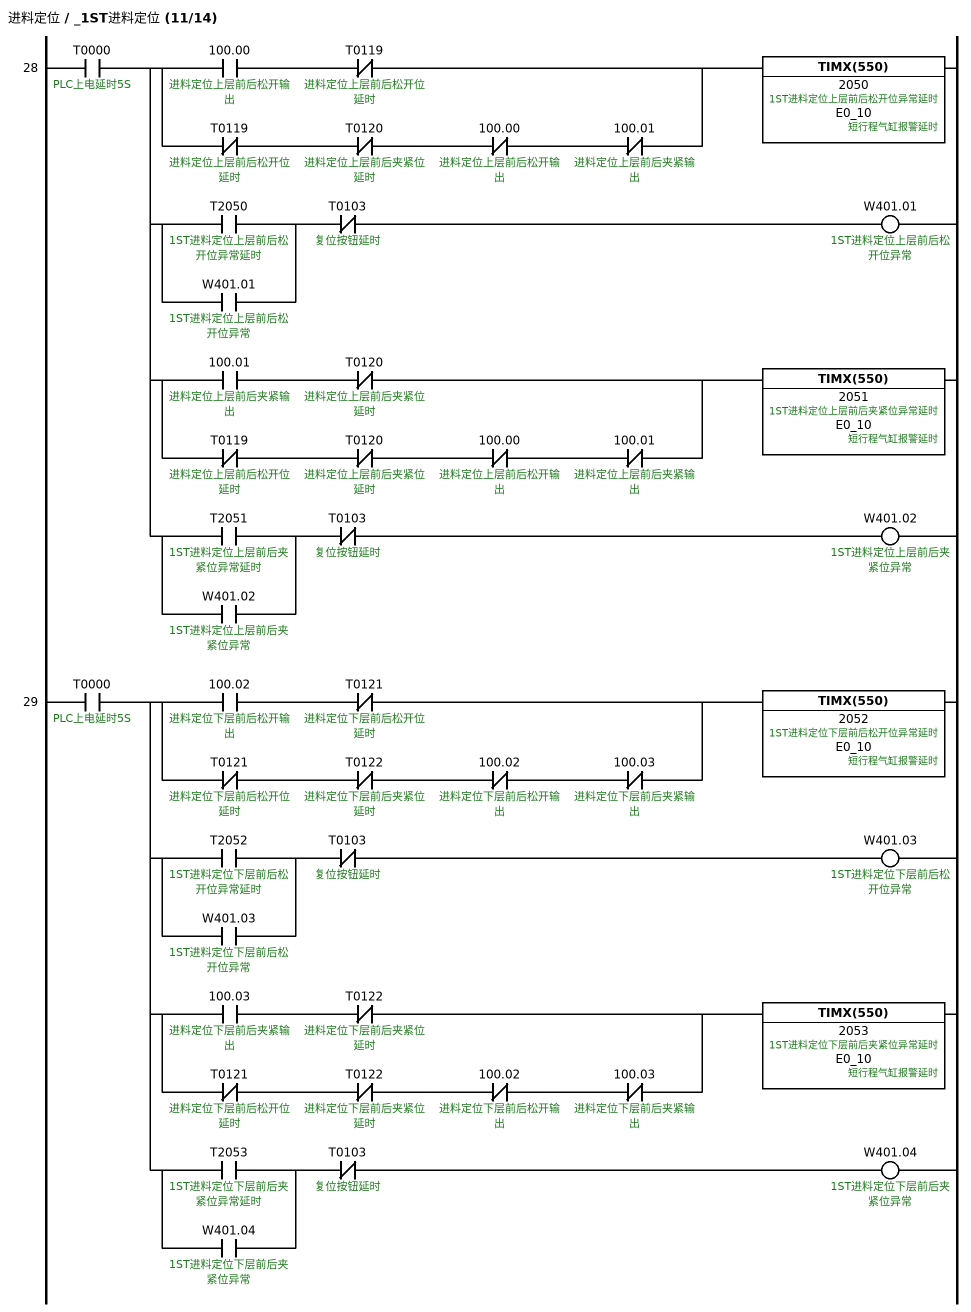
; [picture p72: 进料定位 / _1ST进料定位, rungs 28-29]
; rung 28
LD T0000  ; PLC上电延时5S
OUT TR0
LD 100.00  ; 进料定位上层前后松开输出
ANDNOT T0119  ; 进料定位上层前后松开位延时
LDNOT T0119  ; 进料定位上层前后松开位延时
ANDNOT T0120  ; 进料定位上层前后夹紧位延时
ANDNOT 100.00  ; 进料定位上层前后松开输出
ANDNOT 100.01  ; 进料定位上层前后夹紧输出
ORLD
ANDLD
TIMX(550) 2050 E0_10  ; 短行程气缸报警延时, 1ST进料定位上层前后松开位异常延时
LD TR0
LD T2050  ; 1ST进料定位上层前后松开位异常延时
OR W401.01  ; 1ST进料定位上层前后松开位异常
ANDLD
ANDNOT T0103  ; 复位按钮延时
OUT W401.01  ; 1ST进料定位上层前后松开位异常
LD TR0
LD 100.01  ; 进料定位上层前后夹紧输出
ANDNOT T0120  ; 进料定位上层前后夹紧位延时
LDNOT T0119  ; 进料定位上层前后松开位延时
ANDNOT T0120  ; 进料定位上层前后夹紧位延时
ANDNOT 100.00  ; 进料定位上层前后松开输出
ANDNOT 100.01  ; 进料定位上层前后夹紧输出
ORLD
ANDLD
TIMX(550) 2051 E0_10  ; 短行程气缸报警延时, 1ST进料定位上层前后夹紧位异常延时
LD TR0
LD T2051  ; 1ST进料定位上层前后夹紧位异常延时
OR W401.02  ; 1ST进料定位上层前后夹紧位异常
ANDLD
ANDNOT T0103  ; 复位按钮延时
OUT W401.02  ; 1ST进料定位上层前后夹紧位异常
; rung 29
LD T0000  ; PLC上电延时5S
OUT TR0
LD 100.02  ; 进料定位下层前后松开输出
ANDNOT T0121  ; 进料定位下层前后松开位延时
LDNOT T0121  ; 进料定位下层前后松开位延时
ANDNOT T0122  ; 进料定位下层前后夹紧位延时
ANDNOT 100.02  ; 进料定位下层前后松开输出
ANDNOT 100.03  ; 进料定位下层前后夹紧输出
ORLD
ANDLD
TIMX(550) 2052 E0_10  ; 短行程气缸报警延时, 1ST进料定位下层前后松开位异常延时
LD TR0
LD T2052  ; 1ST进料定位下层前后松开位异常延时
OR W401.03  ; 1ST进料定位下层前后松开位异常
ANDLD
ANDNOT T0103  ; 复位按钮延时
OUT W401.03  ; 1ST进料定位下层前后松开位异常
LD TR0
LD 100.03  ; 进料定位下层前后夹紧输出
ANDNOT T0122  ; 进料定位下层前后夹紧位延时
LDNOT T0121  ; 进料定位下层前后松开位延时
ANDNOT T0122  ; 进料定位下层前后夹紧位延时
ANDNOT 100.02  ; 进料定位下层前后松开输出
ANDNOT 100.03  ; 进料定位下层前后夹紧输出
ORLD
ANDLD
TIMX(550) 2053 E0_10  ; 短行程气缸报警延时, 1ST进料定位下层前后夹紧位异常延时
LD TR0
LD T2053  ; 1ST进料定位下层前后夹紧位异常延时
OR W401.04  ; 1ST进料定位下层前后夹紧位异常
ANDLD
ANDNOT T0103  ; 复位按钮延时
OUT W401.04  ; 1ST进料定位下层前后夹紧位异常

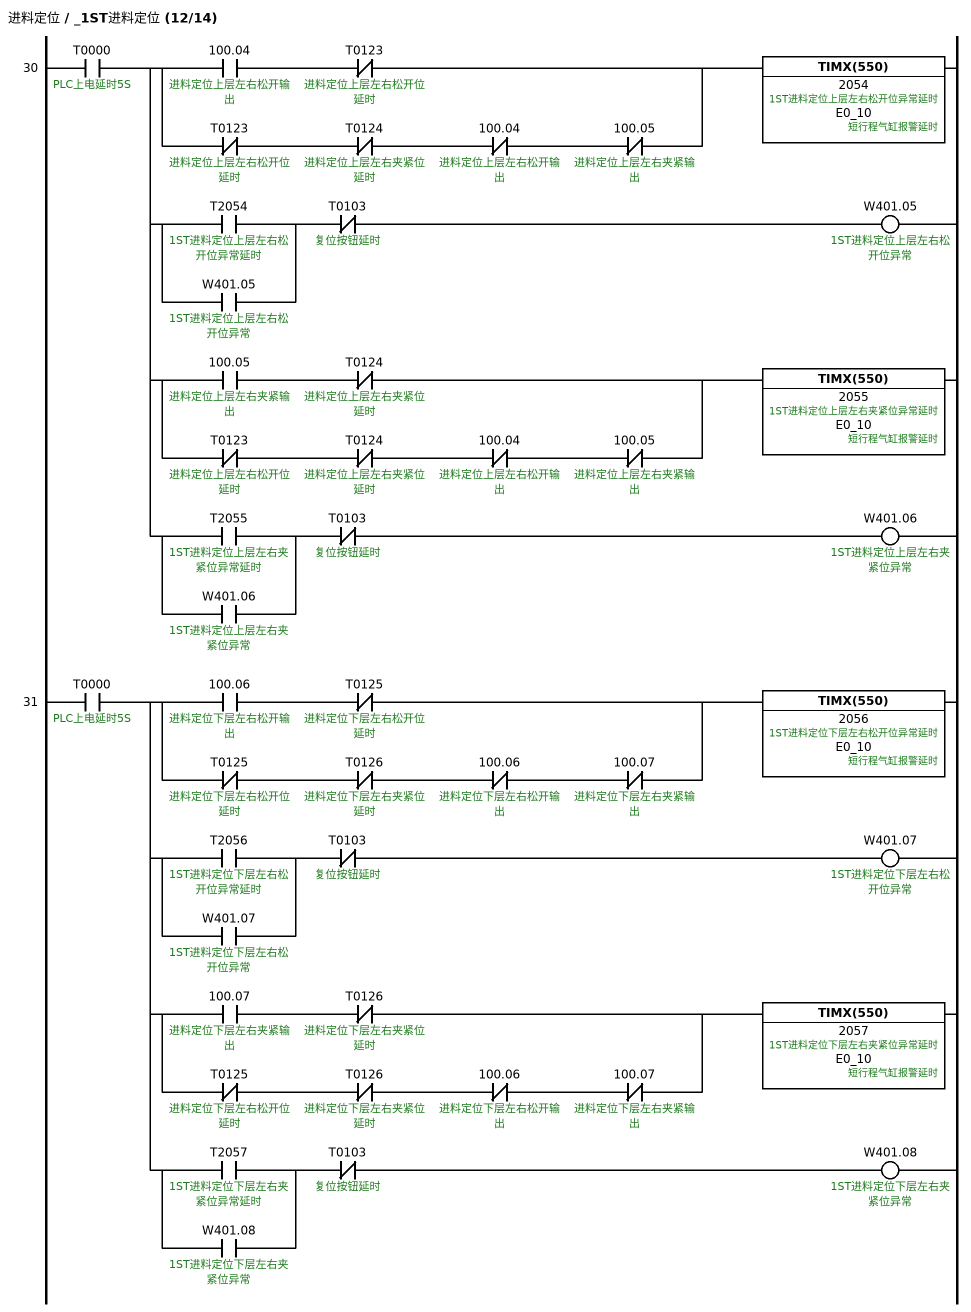
; rung 30
LD T0000  ; PLC上电延时5S
OUT TR0
LD 100.04  ; 进料定位上层左右松开输出
ANDNOT T0123  ; 进料定位上层左右松开位延时
LDNOT T0123  ; 进料定位上层左右松开位延时
ANDNOT T0124  ; 进料定位上层左右夹紧位延时
ANDNOT 100.04  ; 进料定位上层左右松开输出
ANDNOT 100.05  ; 进料定位上层左右夹紧输出
ORLD
ANDLD
TIMX(550) 2054 E0_10  ; 短行程气缸报警延时, 1ST进料定位上层左右松开位异常延时
LD TR0
LD T2054  ; 1ST进料定位上层左右松开位异常延时
OR W401.05  ; 1ST进料定位上层左右松开位异常
ANDLD
ANDNOT T0103  ; 复位按钮延时
OUT W401.05  ; 1ST进料定位上层左右松开位异常
LD TR0
LD 100.05  ; 进料定位上层左右夹紧输出
ANDNOT T0124  ; 进料定位上层左右夹紧位延时
LDNOT T0123  ; 进料定位上层左右松开位延时
ANDNOT T0124  ; 进料定位上层左右夹紧位延时
ANDNOT 100.04  ; 进料定位上层左右松开输出
ANDNOT 100.05  ; 进料定位上层左右夹紧输出
ORLD
ANDLD
TIMX(550) 2055 E0_10  ; 短行程气缸报警延时, 1ST进料定位上层左右夹紧位异常延时
LD TR0
LD T2055  ; 1ST进料定位上层左右夹紧位异常延时
OR W401.06  ; 1ST进料定位上层左右夹紧位异常
ANDLD
ANDNOT T0103  ; 复位按钮延时
OUT W401.06  ; 1ST进料定位上层左右夹紧位异常
; rung 31
LD T0000  ; PLC上电延时5S
OUT TR0
LD 100.06  ; 进料定位下层左右松开输出
ANDNOT T0125  ; 进料定位下层左右松开位延时
LDNOT T0125  ; 进料定位下层左右松开位延时
ANDNOT T0126  ; 进料定位下层左右夹紧位延时
ANDNOT 100.06  ; 进料定位下层左右松开输出
ANDNOT 100.07  ; 进料定位下层左右夹紧输出
ORLD
ANDLD
TIMX(550) 2056 E0_10  ; 短行程气缸报警延时, 1ST进料定位下层左右松开位异常延时
LD TR0
LD T2056  ; 1ST进料定位下层左右松开位异常延时
OR W401.07  ; 1ST进料定位下层左右松开位异常
ANDLD
ANDNOT T0103  ; 复位按钮延时
OUT W401.07  ; 1ST进料定位下层左右松开位异常
LD TR0
LD 100.07  ; 进料定位下层左右夹紧输出
ANDNOT T0126  ; 进料定位下层左右夹紧位延时
LDNOT T0125  ; 进料定位下层左右松开位延时
ANDNOT T0126  ; 进料定位下层左右夹紧位延时
ANDNOT 100.06  ; 进料定位下层左右松开输出
ANDNOT 100.07  ; 进料定位下层左右夹紧输出
ORLD
ANDLD
TIMX(550) 2057 E0_10  ; 短行程气缸报警延时, 1ST进料定位下层左右夹紧位异常延时
LD TR0
LD T2057  ; 1ST进料定位下层左右夹紧位异常延时
OR W401.08  ; 1ST进料定位下层左右夹紧位异常
ANDLD
ANDNOT T0103  ; 复位按钮延时
OUT W401.08  ; 1ST进料定位下层左右夹紧位异常

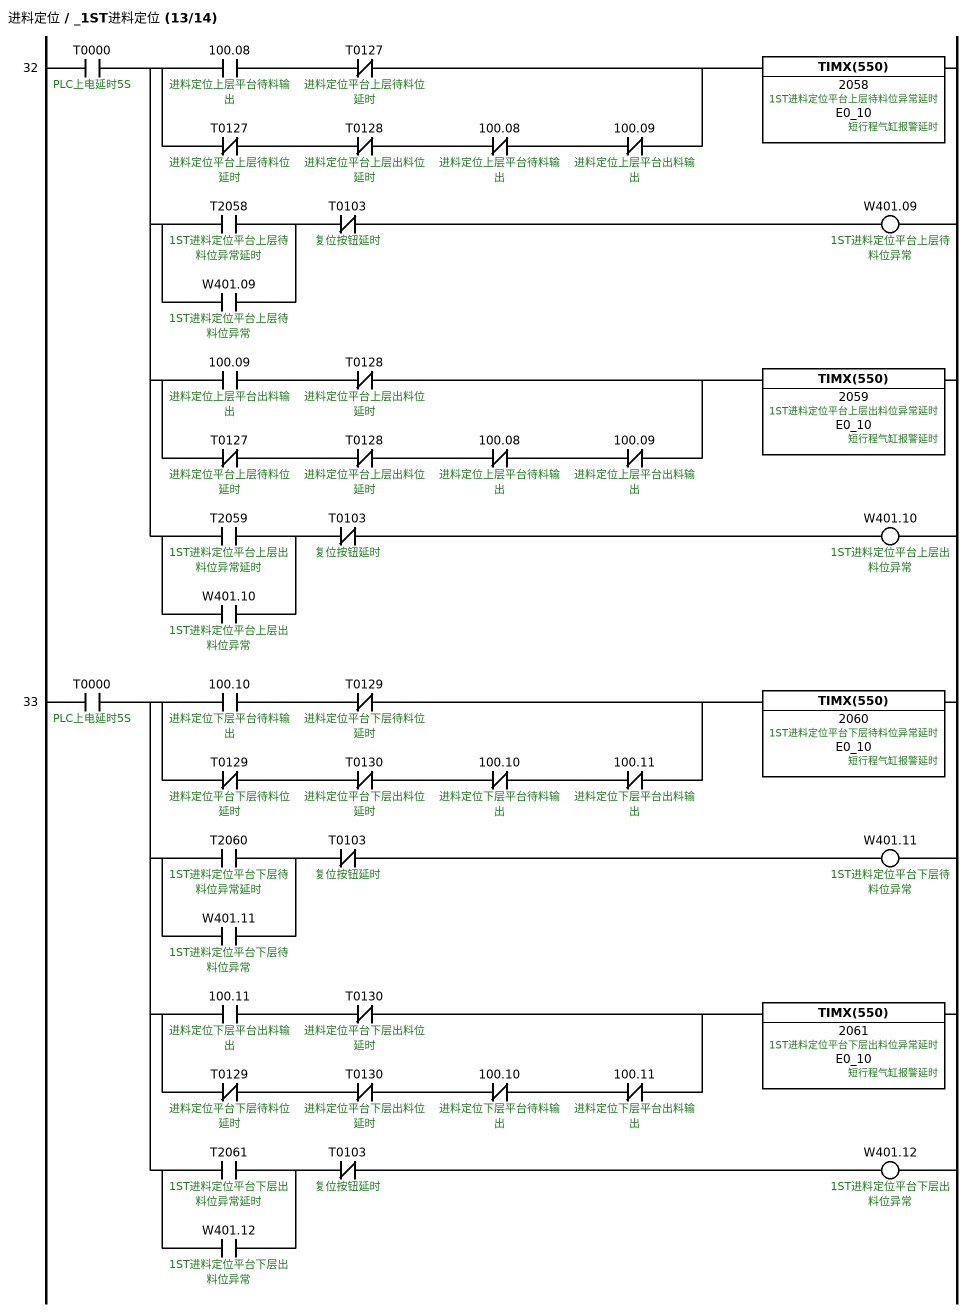
; rung 32
LD T0000  ; PLC上电延时5S
OUT TR0
LD 100.08  ; 进料定位上层平台待料输出
ANDNOT T0127  ; 进料定位平台上层待料位延时
LDNOT T0127  ; 进料定位平台上层待料位延时
ANDNOT T0128  ; 进料定位平台上层出料位延时
ANDNOT 100.08  ; 进料定位上层平台待料输出
ANDNOT 100.09  ; 进料定位上层平台出料输出
ORLD
ANDLD
TIMX(550) 2058 E0_10  ; 短行程气缸报警延时, 1ST进料定位平台上层待料位异常延时
LD TR0
LD T2058  ; 1ST进料定位平台上层待料位异常延时
OR W401.09  ; 1ST进料定位平台上层待料位异常
ANDLD
ANDNOT T0103  ; 复位按钮延时
OUT W401.09  ; 1ST进料定位平台上层待料位异常
LD TR0
LD 100.09  ; 进料定位上层平台出料输出
ANDNOT T0128  ; 进料定位平台上层出料位延时
LDNOT T0127  ; 进料定位平台上层待料位延时
ANDNOT T0128  ; 进料定位平台上层出料位延时
ANDNOT 100.08  ; 进料定位上层平台待料输出
ANDNOT 100.09  ; 进料定位上层平台出料输出
ORLD
ANDLD
TIMX(550) 2059 E0_10  ; 短行程气缸报警延时, 1ST进料定位平台上层出料位异常延时
LD TR0
LD T2059  ; 1ST进料定位平台上层出料位异常延时
OR W401.10  ; 1ST进料定位平台上层出料位异常
ANDLD
ANDNOT T0103  ; 复位按钮延时
OUT W401.10  ; 1ST进料定位平台上层出料位异常
; rung 33
LD T0000  ; PLC上电延时5S
OUT TR0
LD 100.10  ; 进料定位下层平台待料输出
ANDNOT T0129  ; 进料定位平台下层待料位延时
LDNOT T0129  ; 进料定位平台下层待料位延时
ANDNOT T0130  ; 进料定位平台下层出料位延时
ANDNOT 100.10  ; 进料定位下层平台待料输出
ANDNOT 100.11  ; 进料定位下层平台出料输出
ORLD
ANDLD
TIMX(550) 2060 E0_10  ; 短行程气缸报警延时, 1ST进料定位平台下层待料位异常延时
LD TR0
LD T2060  ; 1ST进料定位平台下层待料位异常延时
OR W401.11  ; 1ST进料定位平台下层待料位异常
ANDLD
ANDNOT T0103  ; 复位按钮延时
OUT W401.11  ; 1ST进料定位平台下层待料位异常
LD TR0
LD 100.11  ; 进料定位下层平台出料输出
ANDNOT T0130  ; 进料定位平台下层出料位延时
LDNOT T0129  ; 进料定位平台下层待料位延时
ANDNOT T0130  ; 进料定位平台下层出料位延时
ANDNOT 100.10  ; 进料定位下层平台待料输出
ANDNOT 100.11  ; 进料定位下层平台出料输出
ORLD
ANDLD
TIMX(550) 2061 E0_10  ; 短行程气缸报警延时, 1ST进料定位平台下层出料位异常延时
LD TR0
LD T2061  ; 1ST进料定位平台下层出料位异常延时
OR W401.12  ; 1ST进料定位平台下层出料位异常
ANDLD
ANDNOT T0103  ; 复位按钮延时
OUT W401.12  ; 1ST进料定位平台下层出料位异常

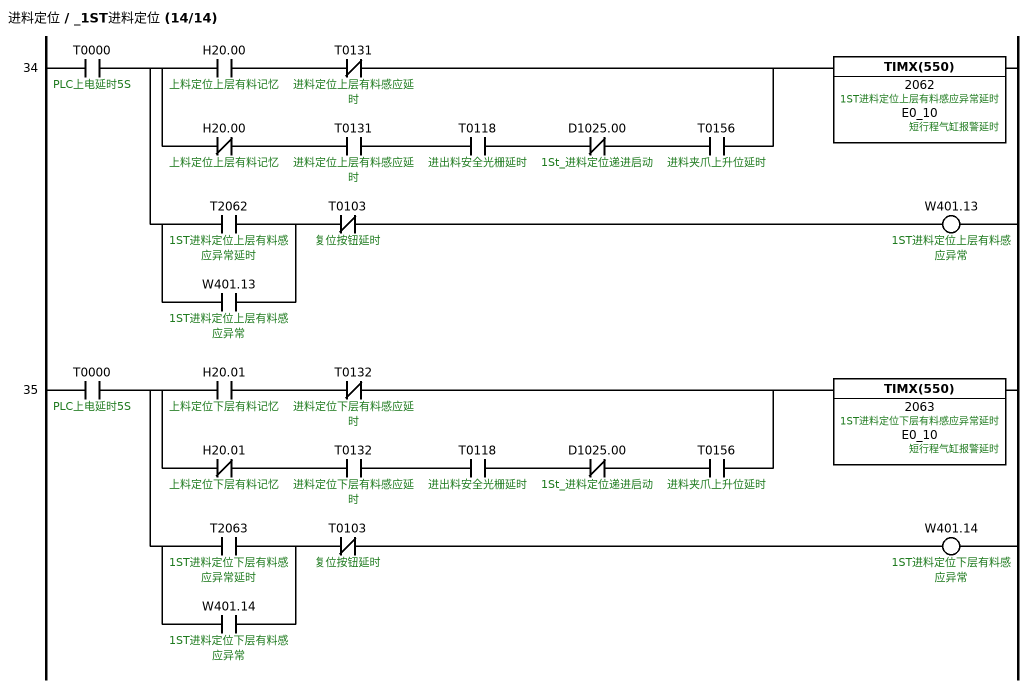
; rung 34
LD T0000  ; PLC上电延时5S
OUT TR0
LD H20.00  ; 上料定位上层有料记忆
ANDNOT T0131  ; 进料定位上层有料感应延时
LDNOT H20.00  ; 上料定位上层有料记忆
AND T0131  ; 进料定位上层有料感应延时
AND T0118  ; 进出料安全光栅延时
ANDNOT D1025.00  ; 1St_进料定位递进启动
AND T0156  ; 进料夹爪上升位延时
ORLD
ANDLD
TIMX(550) 2062 E0_10  ; 短行程气缸报警延时, 1ST进料定位上层有料感应异常延时
LD TR0
LD T2062  ; 1ST进料定位上层有料感应异常延时
OR W401.13  ; 1ST进料定位上层有料感应异常
ANDLD
ANDNOT T0103  ; 复位按钮延时
OUT W401.13  ; 1ST进料定位上层有料感应异常
; rung 35
LD T0000  ; PLC上电延时5S
OUT TR0
LD H20.01  ; 上料定位下层有料记忆
ANDNOT T0132  ; 进料定位下层有料感应延时
LDNOT H20.01  ; 上料定位下层有料记忆
AND T0132  ; 进料定位下层有料感应延时
AND T0118  ; 进出料安全光栅延时
ANDNOT D1025.00  ; 1St_进料定位递进启动
AND T0156  ; 进料夹爪上升位延时
ORLD
ANDLD
TIMX(550) 2063 E0_10  ; 短行程气缸报警延时, 1ST进料定位下层有料感应异常延时
LD TR0
LD T2063  ; 1ST进料定位下层有料感应异常延时
OR W401.14  ; 1ST进料定位下层有料感应异常
ANDLD
ANDNOT T0103  ; 复位按钮延时
OUT W401.14  ; 1ST进料定位下层有料感应异常

### Section 复位

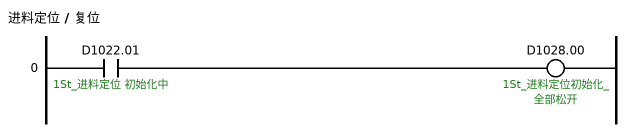
; rung 0
LD D1022.01  ; 1St_进料定位 初始化中
OUT D1028.00  ; 1St_进料定位初始化_全部松开

### Section 输出

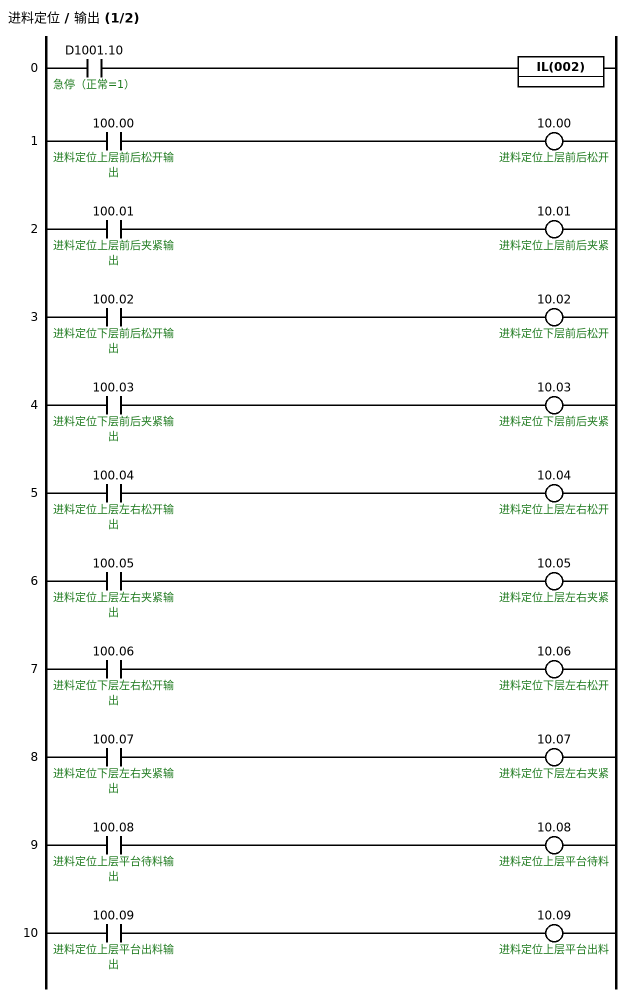
; rung 0
LD D1001.10  ; 急停（正常=1）
IL(002)
; rung 1
LD 100.00  ; 进料定位上层前后松开输出
OUT 10.00  ; 进料定位上层前后松开
; rung 2
LD 100.01  ; 进料定位上层前后夹紧输出
OUT 10.01  ; 进料定位上层前后夹紧
; rung 3
LD 100.02  ; 进料定位下层前后松开输出
OUT 10.02  ; 进料定位下层前后松开
; rung 4
LD 100.03  ; 进料定位下层前后夹紧输出
OUT 10.03  ; 进料定位下层前后夹紧
; rung 5
LD 100.04  ; 进料定位上层左右松开输出
OUT 10.04  ; 进料定位上层左右松开
; rung 6
LD 100.05  ; 进料定位上层左右夹紧输出
OUT 10.05  ; 进料定位上层左右夹紧
; rung 7
LD 100.06  ; 进料定位下层左右松开输出
OUT 10.06  ; 进料定位下层左右松开
; rung 8
LD 100.07  ; 进料定位下层左右夹紧输出
OUT 10.07  ; 进料定位下层左右夹紧
; rung 9
LD 100.08  ; 进料定位上层平台待料输出
OUT 10.08  ; 进料定位上层平台待料
; rung 10
LD 100.09  ; 进料定位上层平台出料输出
OUT 10.09  ; 进料定位上层平台出料

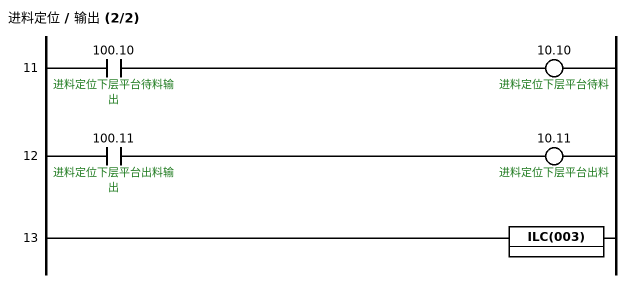
; rung 11
LD 100.10  ; 进料定位下层平台待料输出
OUT 10.10  ; 进料定位下层平台待料
; rung 12
LD 100.11  ; 进料定位下层平台出料输出
OUT 10.11  ; 进料定位下层平台出料
; rung 13
ILC(003)

### Section END
; rung 0
END(001)

## Program 出料定位 (cyclic task 2)

### Section Main

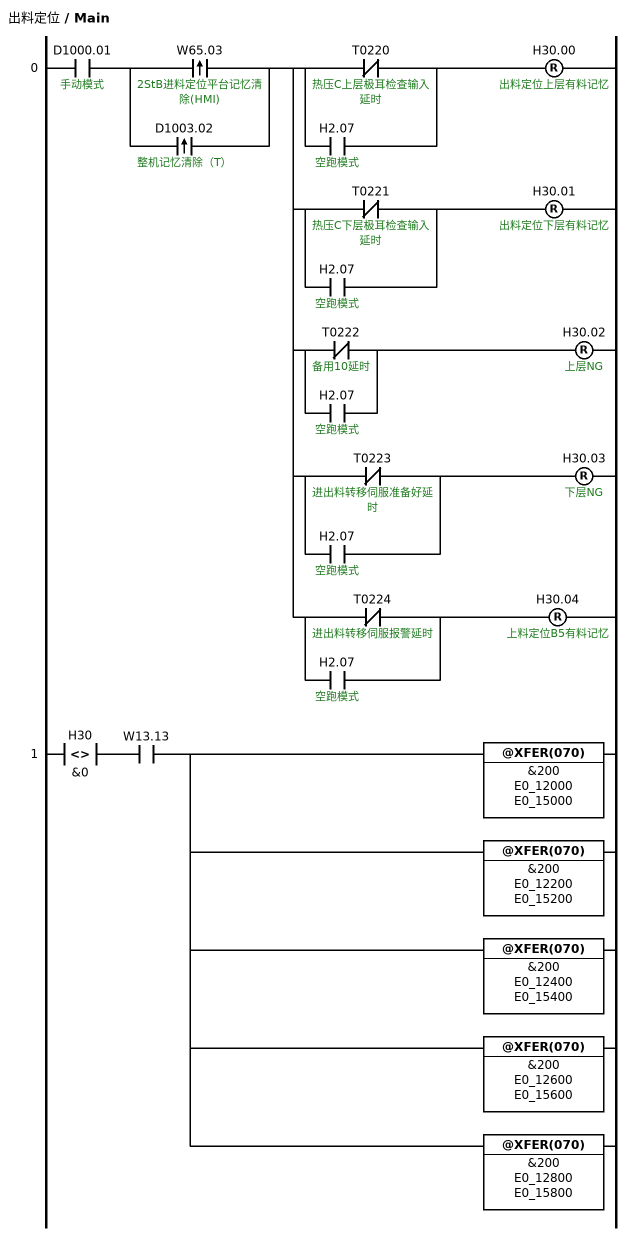
; rung 0
LD D1000.01  ; 手动模式
@LD W65.03  ; 2StB进料定位平台记忆清除(HMI)
@OR D1003.02  ; 整机记忆清除（T）
ANDLD
OUT TR0
LDNOT T0220  ; 热压C上层极耳检查输入延时
OR H2.07  ; 空跑模式
ANDLD
RSET H30.00  ; 出料定位上层有料记忆
LD TR0
LDNOT T0221  ; 热压C下层极耳检查输入延时
OR H2.07  ; 空跑模式
ANDLD
RSET H30.01  ; 出料定位下层有料记忆
LD TR0
LDNOT T0222  ; 备用10延时
OR H2.07  ; 空跑模式
ANDLD
RSET H30.02  ; 上层NG
LD TR0
LDNOT T0223  ; 进出料转移伺服准备好延时
OR H2.07  ; 空跑模式
ANDLD
RSET H30.03  ; 下层NG
LD TR0
LDNOT T0224  ; 进出料转移伺服报警延时
OR H2.07  ; 空跑模式
ANDLD
RSET H30.04  ; 上料定位B5有料记忆
; rung 1
LD<>(305) H30 &0
AND W13.13
@XFER(070) &200 E0_12000 E0_15000
@XFER(070) &200 E0_12200 E0_15200
@XFER(070) &200 E0_12400 E0_15400
@XFER(070) &200 E0_12600 E0_15600
@XFER(070) &200 E0_12800 E0_15800

### Section _2ST出料定位

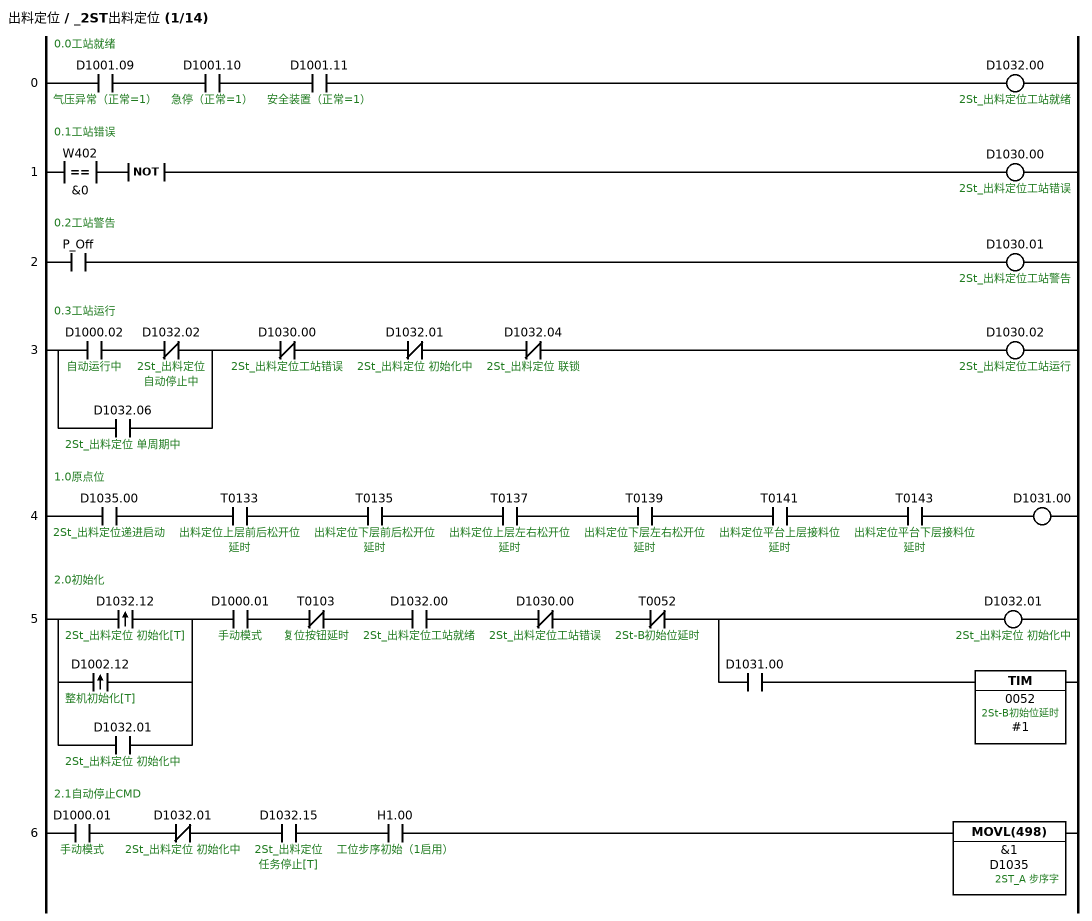
; rung 0: 0.0工站就绪
LD D1001.09  ; 气压异常（正常=1）
AND D1001.10  ; 急停（正常=1）
AND D1001.11  ; 安全装置（正常=1）
OUT D1032.00  ; 2St_出料定位工站就绪
; rung 1: 0.1工站错误
LD=(300) W402 &0
NOT(520)
OUT D1030.00  ; 2St_出料定位工站错误
; rung 2: 0.2工站警告
LD P_Off
OUT D1030.01  ; 2St_出料定位工站警告
; rung 3: 0.3工站运行
LD D1000.02  ; 自动运行中
ANDNOT D1032.02  ; 2St_出料定位 自动停止中
OR D1032.06  ; 2St_出料定位 单周期中
ANDNOT D1030.00  ; 2St_出料定位工站错误
ANDNOT D1032.01  ; 2St_出料定位 初始化中
ANDNOT D1032.04  ; 2St_出料定位 联锁
OUT D1030.02  ; 2St_出料定位工站运行
; rung 4: 1.0原点位
LD D1035.00  ; 2St_出料定位递进启动
AND T0133  ; 出料定位上层前后松开位延时
AND T0135  ; 出料定位下层前后松开位延时
AND T0137  ; 出料定位上层左右松开位延时
AND T0139  ; 出料定位下层左右松开位延时
AND T0141  ; 出料定位平台上层接料位延时
AND T0143  ; 出料定位平台下层接料位延时
OUT D1031.00
; rung 5: 2.0初始化
@LD D1032.12  ; 2St_出料定位 初始化[T]
@OR D1002.12  ; 整机初始化[T]
OR D1032.01  ; 2St_出料定位 初始化中
AND D1000.01  ; 手动模式
ANDNOT T0103  ; 复位按钮延时
AND D1032.00  ; 2St_出料定位工站就绪
ANDNOT D1030.00  ; 2St_出料定位工站错误
ANDNOT T0052  ; 2St-B初始位延时
OUT D1032.01  ; 2St_出料定位 初始化中
AND D1031.00
TIM 0052 #1  ; 2St-B初始位延时
; rung 6: 2.1自动停止CMD
LD D1000.01  ; 手动模式
ANDNOT D1032.01  ; 2St_出料定位 初始化中
AND D1032.15  ; 2St_出料定位 任务停止[T]
AND H1.00  ; 工位步序初始（1启用）
MOVL(498) &1 D1035  ; 2ST_A 步序字

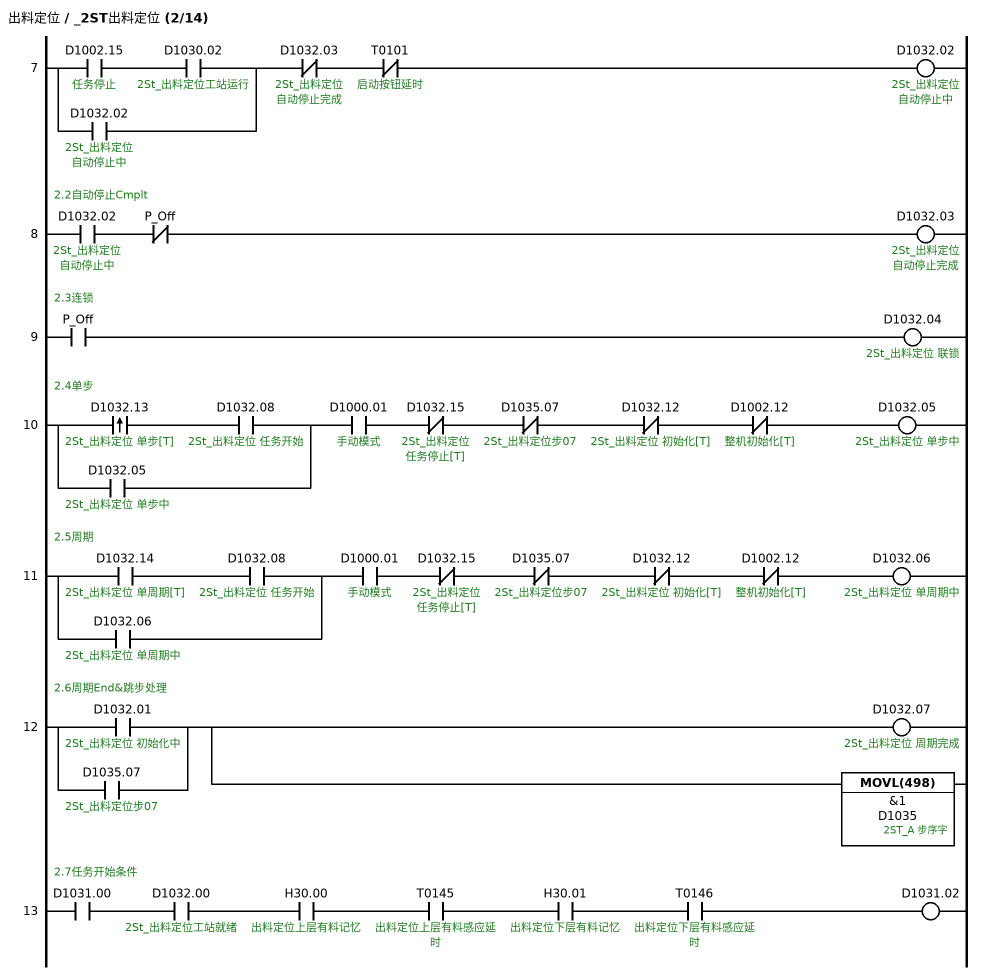
; rung 7
LD D1002.15  ; 任务停止
AND D1030.02  ; 2St_出料定位工站运行
OR D1032.02  ; 2St_出料定位 自动停止中
ANDNOT D1032.03  ; 2St_出料定位 自动停止完成
ANDNOT T0101  ; 启动按钮延时
OUT D1032.02  ; 2St_出料定位 自动停止中
; rung 8: 2.2自动停止Cmplt
LD D1032.02  ; 2St_出料定位 自动停止中
ANDNOT P_Off
OUT D1032.03  ; 2St_出料定位 自动停止完成
; rung 9: 2.3连锁
LD P_Off
OUT D1032.04  ; 2St_出料定位 联锁
; rung 10: 2.4单步
@LD D1032.13  ; 2St_出料定位 单步[T]
AND D1032.08  ; 2St_出料定位 任务开始
OR D1032.05  ; 2St_出料定位 单步中
AND D1000.01  ; 手动模式
ANDNOT D1032.15  ; 2St_出料定位 任务停止[T]
ANDNOT D1035.07  ; 2St_出料定位步07
ANDNOT D1032.12  ; 2St_出料定位 初始化[T]
ANDNOT D1002.12  ; 整机初始化[T]
OUT D1032.05  ; 2St_出料定位 单步中
; rung 11: 2.5周期
LD D1032.14  ; 2St_出料定位 单周期[T]
AND D1032.08  ; 2St_出料定位 任务开始
OR D1032.06  ; 2St_出料定位 单周期中
AND D1000.01  ; 手动模式
ANDNOT D1032.15  ; 2St_出料定位 任务停止[T]
ANDNOT D1035.07  ; 2St_出料定位步07
ANDNOT D1032.12  ; 2St_出料定位 初始化[T]
ANDNOT D1002.12  ; 整机初始化[T]
OUT D1032.06  ; 2St_出料定位 单周期中
; rung 12: 2.6周期End&跳步处理
LD D1032.01  ; 2St_出料定位 初始化中
OR D1035.07  ; 2St_出料定位步07
OUT D1032.07  ; 2St_出料定位 周期完成
MOVL(498) &1 D1035  ; 2ST_A 步序字
; rung 13: 2.7任务开始条件
LD D1031.00
AND D1032.00  ; 2St_出料定位工站就绪
AND H30.00  ; 出料定位上层有料记忆
AND T0145  ; 出料定位上层有料感应延时
AND H30.01  ; 出料定位下层有料记忆
AND T0146  ; 出料定位下层有料感应延时
OUT D1031.02

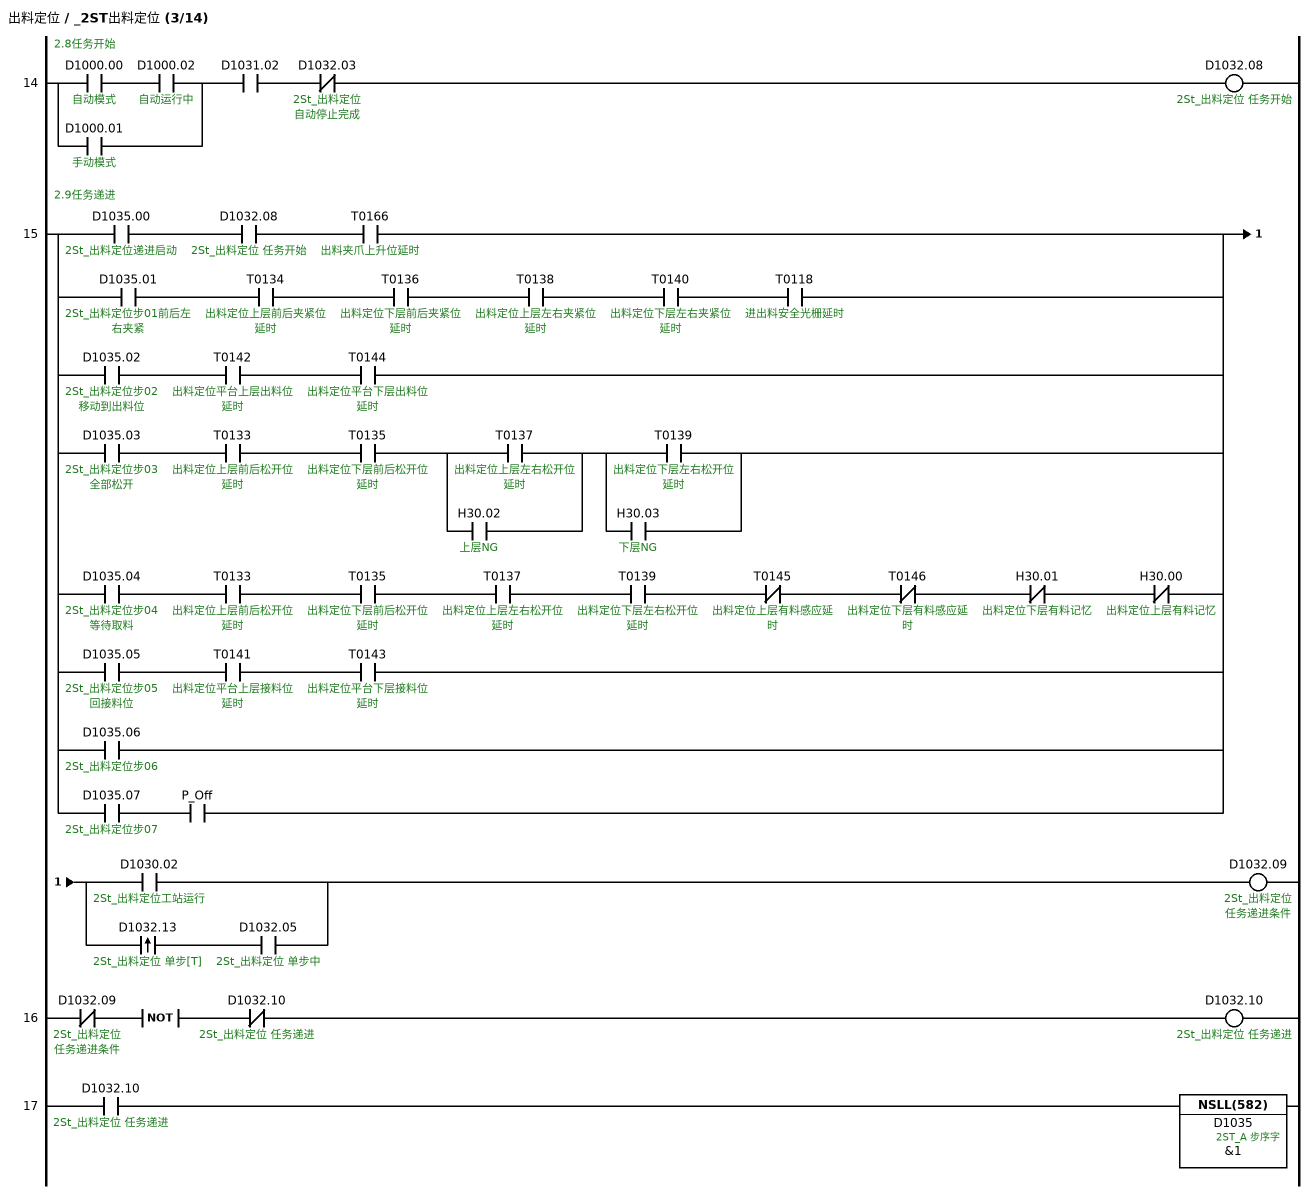
; rung 14: 2.8任务开始
LD D1000.00  ; 自动模式
AND D1000.02  ; 自动运行中
OR D1000.01  ; 手动模式
AND D1031.02
ANDNOT D1032.03  ; 2St_出料定位 自动停止完成
OUT D1032.08  ; 2St_出料定位 任务开始
; rung 15: 2.9任务递进
LD D1035.00  ; 2St_出料定位递进启动
AND D1032.08  ; 2St_出料定位 任务开始
AND T0166  ; 出料夹爪上升位延时
LD D1035.01  ; 2St_出料定位步01前后左右夹紧
AND T0134  ; 出料定位上层前后夹紧位延时
AND T0136  ; 出料定位下层前后夹紧位延时
AND T0138  ; 出料定位上层左右夹紧位延时
AND T0140  ; 出料定位下层左右夹紧位延时
AND T0118  ; 进出料安全光栅延时
ORLD
LD D1035.02  ; 2St_出料定位步02 移动到出料位
AND T0142  ; 出料定位平台上层出料位延时
AND T0144  ; 出料定位平台下层出料位延时
ORLD
LD D1035.03  ; 2St_出料定位步03 全部松开
AND T0133  ; 出料定位上层前后松开位延时
AND T0135  ; 出料定位下层前后松开位延时
LD T0137  ; 出料定位上层左右松开位延时
OR H30.02  ; 上层NG
ANDLD
LD T0139  ; 出料定位下层左右松开位延时
OR H30.03  ; 下层NG
ANDLD
ORLD
LD D1035.04  ; 2St_出料定位步04 等待取料
AND T0133  ; 出料定位上层前后松开位延时
AND T0135  ; 出料定位下层前后松开位延时
AND T0137  ; 出料定位上层左右松开位延时
AND T0139  ; 出料定位下层左右松开位延时
ANDNOT T0145  ; 出料定位上层有料感应延时
ANDNOT T0146  ; 出料定位下层有料感应延时
ANDNOT H30.01  ; 出料定位下层有料记忆
ANDNOT H30.00  ; 出料定位上层有料记忆
ORLD
LD D1035.05  ; 2St_出料定位步05 回接料位
AND T0141  ; 出料定位平台上层接料位延时
AND T0143  ; 出料定位平台下层接料位延时
ORLD
OR D1035.06  ; 2St_出料定位步06
LD D1035.07  ; 2St_出料定位步07
AND P_Off
ORLD
LD D1030.02  ; 2St_出料定位工站运行
@LD D1032.13  ; 2St_出料定位 单步[T]
AND D1032.05  ; 2St_出料定位 单步中
ORLD
ANDLD
OUT D1032.09  ; 2St_出料定位 任务递进条件
; rung 16
LDNOT D1032.09  ; 2St_出料定位 任务递进条件
NOT(520)
ANDNOT D1032.10  ; 2St_出料定位 任务递进
OUT D1032.10  ; 2St_出料定位 任务递进
; rung 17
LD D1032.10  ; 2St_出料定位 任务递进
NSLL(582) D1035 &1  ; 2ST_A 步序字

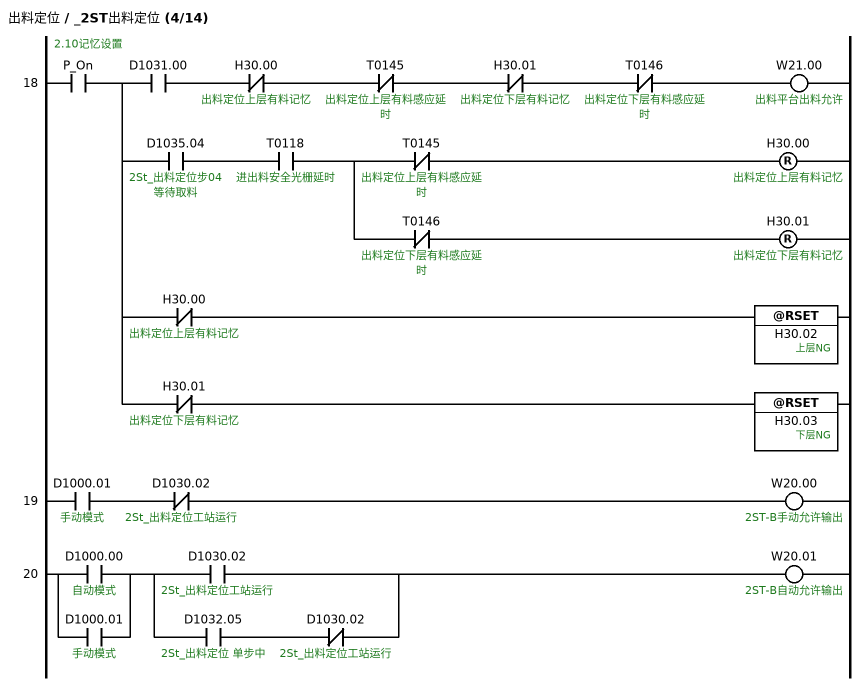
; rung 18: 2.10记忆设置
LD P_On
OUT TR0
AND D1031.00
ANDNOT H30.00  ; 出料定位上层有料记忆
ANDNOT T0145  ; 出料定位上层有料感应延时
ANDNOT H30.01  ; 出料定位下层有料记忆
ANDNOT T0146  ; 出料定位下层有料感应延时
OUT W21.00  ; 出料平台出料允许
LD TR0
AND D1035.04  ; 2St_出料定位步04 等待取料
AND T0118  ; 进出料安全光栅延时
OUT TR1
ANDNOT T0145  ; 出料定位上层有料感应延时
RSET H30.00  ; 出料定位上层有料记忆
LD TR1
ANDNOT T0146  ; 出料定位下层有料感应延时
RSET H30.01  ; 出料定位下层有料记忆
LD TR0
ANDNOT H30.00  ; 出料定位上层有料记忆
@RSET H30.02  ; 上层NG
LD TR0
ANDNOT H30.01  ; 出料定位下层有料记忆
@RSET H30.03  ; 下层NG
; rung 19
LD D1000.01  ; 手动模式
ANDNOT D1030.02  ; 2St_出料定位工站运行
OUT W20.00  ; 2ST-B手动允许输出
; rung 20
LD D1000.00  ; 自动模式
OR D1000.01  ; 手动模式
LD D1030.02  ; 2St_出料定位工站运行
LD D1032.05  ; 2St_出料定位 单步中
ANDNOT D1030.02  ; 2St_出料定位工站运行
ORLD
ANDLD
OUT W20.01  ; 2ST-B自动允许输出

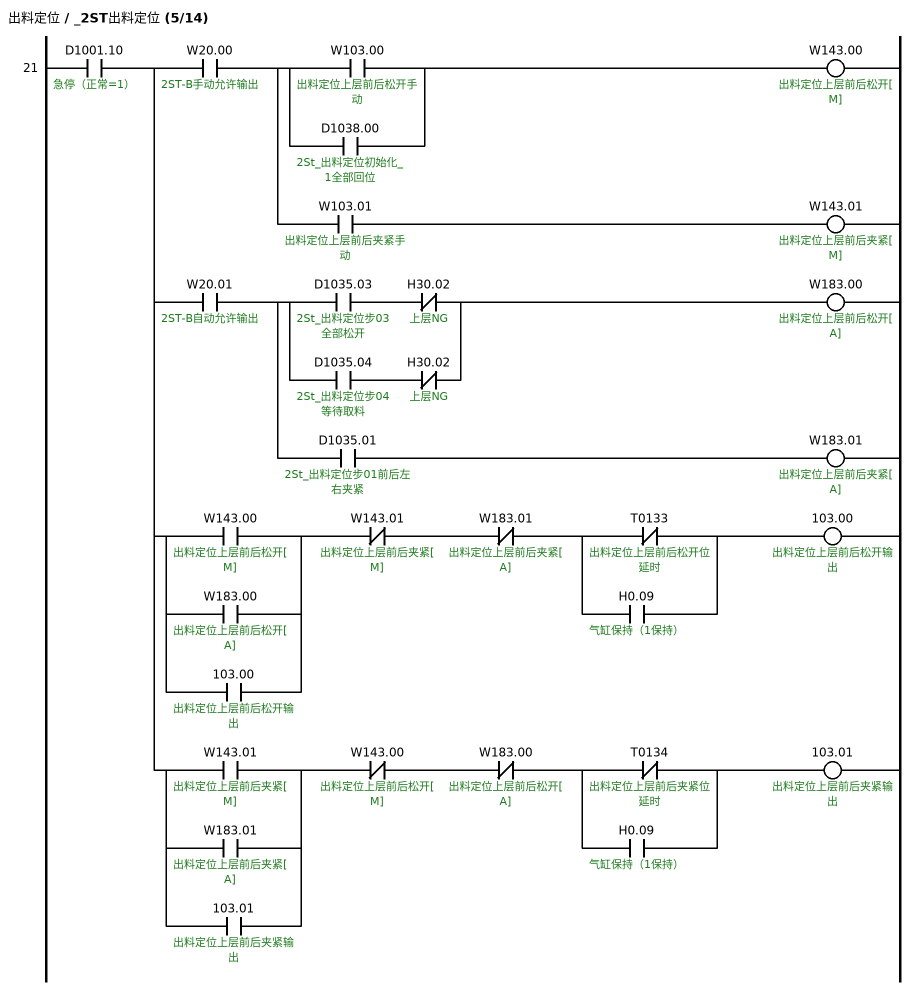
; rung 21
LD D1001.10  ; 急停（正常=1）
OUT TR0
AND W20.00  ; 2ST-B手动允许输出
OUT TR1
LD W103.00  ; 出料定位上层前后松开手动
OR D1038.00  ; 2St_出料定位初始化_1全部回位
ANDLD
OUT W143.00  ; 出料定位上层前后松开[M]
LD TR1
AND W103.01  ; 出料定位上层前后夹紧手动
OUT W143.01  ; 出料定位上层前后夹紧[M]
LD TR0
AND W20.01  ; 2ST-B自动允许输出
OUT TR1
LD D1035.03  ; 2St_出料定位步03 全部松开
ANDNOT H30.02  ; 上层NG
LD D1035.04  ; 2St_出料定位步04 等待取料
ANDNOT H30.02  ; 上层NG
ORLD
ANDLD
OUT W183.00  ; 出料定位上层前后松开[A]
LD TR1
AND D1035.01  ; 2St_出料定位步01前后左右夹紧
OUT W183.01  ; 出料定位上层前后夹紧[A]
LD TR0
LD W143.00  ; 出料定位上层前后松开[M]
OR W183.00  ; 出料定位上层前后松开[A]
OR 103.00  ; 出料定位上层前后松开输出
ANDLD
ANDNOT W143.01  ; 出料定位上层前后夹紧[M]
ANDNOT W183.01  ; 出料定位上层前后夹紧[A]
LDNOT T0133  ; 出料定位上层前后松开位延时
OR H0.09  ; 气缸保持（1保持）
ANDLD
OUT 103.00  ; 出料定位上层前后松开输出
LD TR0
LD W143.01  ; 出料定位上层前后夹紧[M]
OR W183.01  ; 出料定位上层前后夹紧[A]
OR 103.01  ; 出料定位上层前后夹紧输出
ANDLD
ANDNOT W143.00  ; 出料定位上层前后松开[M]
ANDNOT W183.00  ; 出料定位上层前后松开[A]
LDNOT T0134  ; 出料定位上层前后夹紧位延时
OR H0.09  ; 气缸保持（1保持）
ANDLD
OUT 103.01  ; 出料定位上层前后夹紧输出

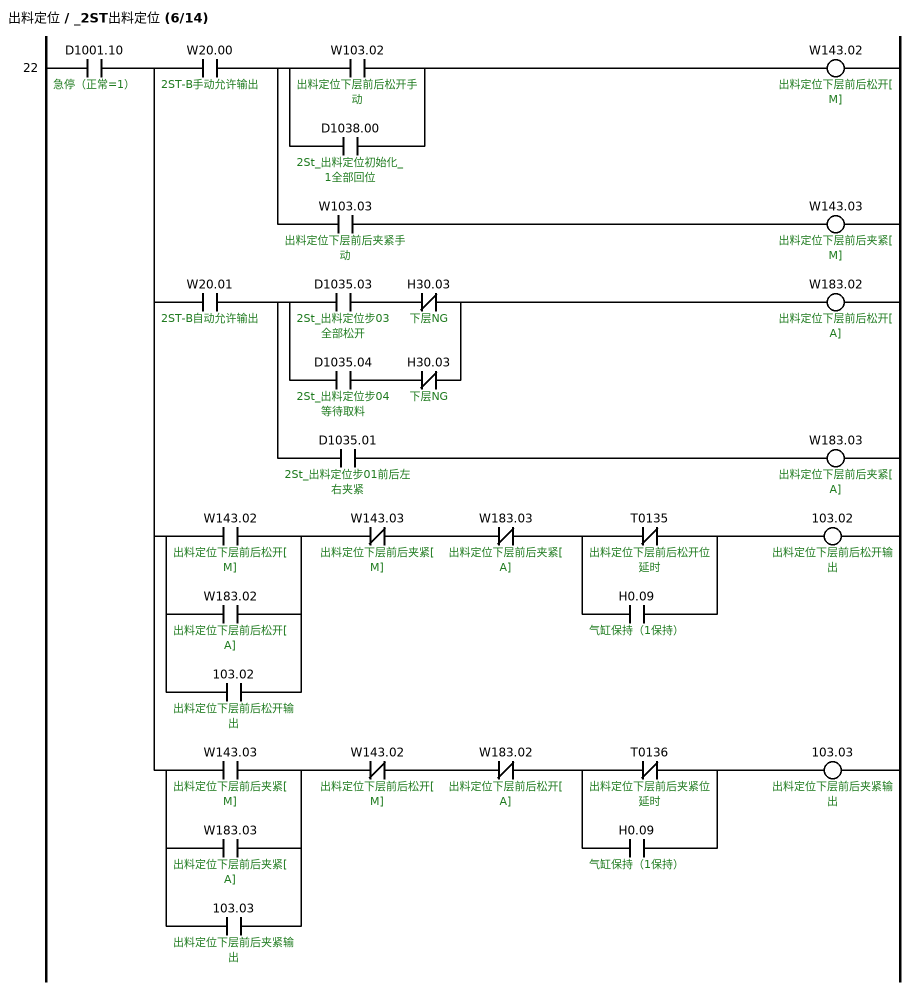
; rung 22
LD D1001.10  ; 急停（正常=1）
OUT TR0
AND W20.00  ; 2ST-B手动允许输出
OUT TR1
LD W103.02  ; 出料定位下层前后松开手动
OR D1038.00  ; 2St_出料定位初始化_1全部回位
ANDLD
OUT W143.02  ; 出料定位下层前后松开[M]
LD TR1
AND W103.03  ; 出料定位下层前后夹紧手动
OUT W143.03  ; 出料定位下层前后夹紧[M]
LD TR0
AND W20.01  ; 2ST-B自动允许输出
OUT TR1
LD D1035.03  ; 2St_出料定位步03 全部松开
ANDNOT H30.03  ; 下层NG
LD D1035.04  ; 2St_出料定位步04 等待取料
ANDNOT H30.03  ; 下层NG
ORLD
ANDLD
OUT W183.02  ; 出料定位下层前后松开[A]
LD TR1
AND D1035.01  ; 2St_出料定位步01前后左右夹紧
OUT W183.03  ; 出料定位下层前后夹紧[A]
LD TR0
LD W143.02  ; 出料定位下层前后松开[M]
OR W183.02  ; 出料定位下层前后松开[A]
OR 103.02  ; 出料定位下层前后松开输出
ANDLD
ANDNOT W143.03  ; 出料定位下层前后夹紧[M]
ANDNOT W183.03  ; 出料定位下层前后夹紧[A]
LDNOT T0135  ; 出料定位下层前后松开位延时
OR H0.09  ; 气缸保持（1保持）
ANDLD
OUT 103.02  ; 出料定位下层前后松开输出
LD TR0
LD W143.03  ; 出料定位下层前后夹紧[M]
OR W183.03  ; 出料定位下层前后夹紧[A]
OR 103.03  ; 出料定位下层前后夹紧输出
ANDLD
ANDNOT W143.02  ; 出料定位下层前后松开[M]
ANDNOT W183.02  ; 出料定位下层前后松开[A]
LDNOT T0136  ; 出料定位下层前后夹紧位延时
OR H0.09  ; 气缸保持（1保持）
ANDLD
OUT 103.03  ; 出料定位下层前后夹紧输出

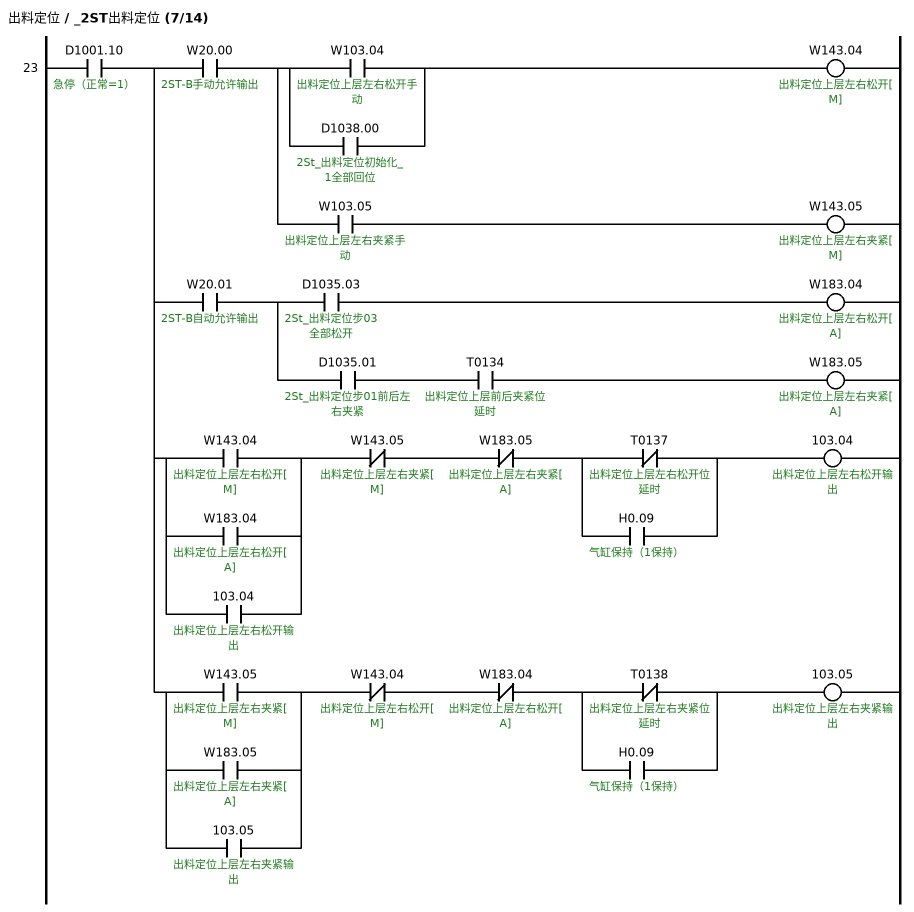
; rung 23
LD D1001.10  ; 急停（正常=1）
OUT TR0
AND W20.00  ; 2ST-B手动允许输出
OUT TR1
LD W103.04  ; 出料定位上层左右松开手动
OR D1038.00  ; 2St_出料定位初始化_1全部回位
ANDLD
OUT W143.04  ; 出料定位上层左右松开[M]
LD TR1
AND W103.05  ; 出料定位上层左右夹紧手动
OUT W143.05  ; 出料定位上层左右夹紧[M]
LD TR0
AND W20.01  ; 2ST-B自动允许输出
OUT TR1
AND D1035.03  ; 2St_出料定位步03 全部松开
OUT W183.04  ; 出料定位上层左右松开[A]
LD TR1
AND D1035.01  ; 2St_出料定位步01前后左右夹紧
AND T0134  ; 出料定位上层前后夹紧位延时
OUT W183.05  ; 出料定位上层左右夹紧[A]
LD TR0
LD W143.04  ; 出料定位上层左右松开[M]
OR W183.04  ; 出料定位上层左右松开[A]
OR 103.04  ; 出料定位上层左右松开输出
ANDLD
ANDNOT W143.05  ; 出料定位上层左右夹紧[M]
ANDNOT W183.05  ; 出料定位上层左右夹紧[A]
LDNOT T0137  ; 出料定位上层左右松开位延时
OR H0.09  ; 气缸保持（1保持）
ANDLD
OUT 103.04  ; 出料定位上层左右松开输出
LD TR0
LD W143.05  ; 出料定位上层左右夹紧[M]
OR W183.05  ; 出料定位上层左右夹紧[A]
OR 103.05  ; 出料定位上层左右夹紧输出
ANDLD
ANDNOT W143.04  ; 出料定位上层左右松开[M]
ANDNOT W183.04  ; 出料定位上层左右松开[A]
LDNOT T0138  ; 出料定位上层左右夹紧位延时
OR H0.09  ; 气缸保持（1保持）
ANDLD
OUT 103.05  ; 出料定位上层左右夹紧输出

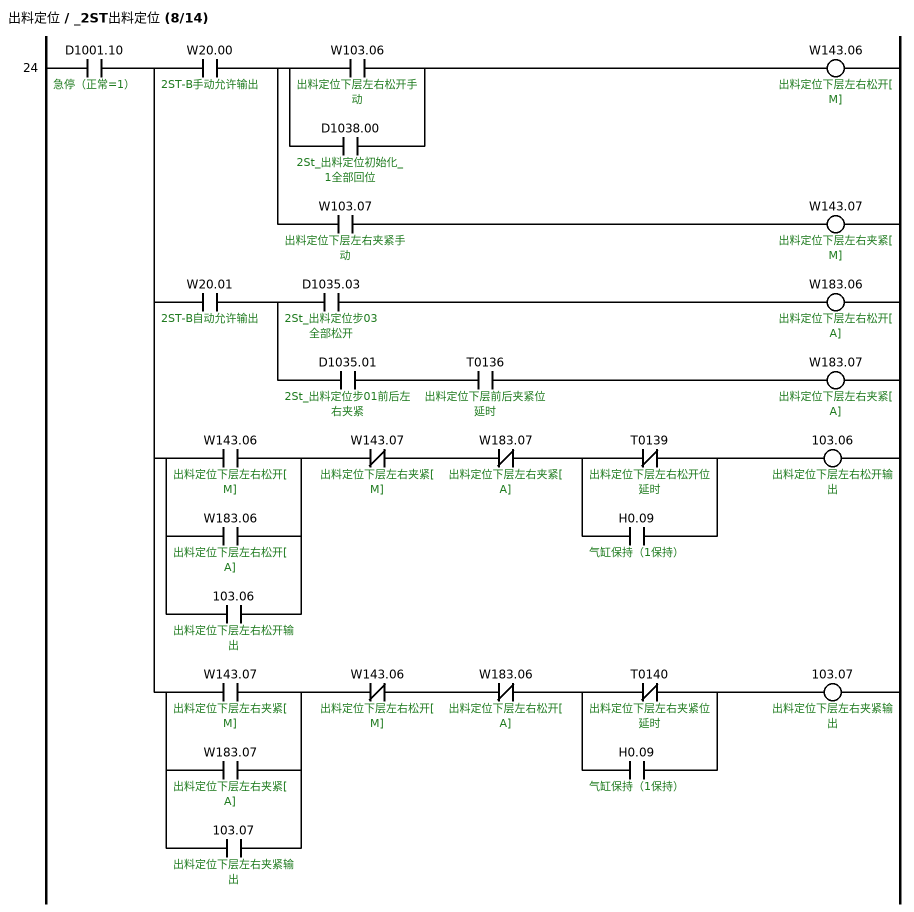
; rung 24
LD D1001.10  ; 急停（正常=1）
OUT TR0
AND W20.00  ; 2ST-B手动允许输出
OUT TR1
LD W103.06  ; 出料定位下层左右松开手动
OR D1038.00  ; 2St_出料定位初始化_1全部回位
ANDLD
OUT W143.06  ; 出料定位下层左右松开[M]
LD TR1
AND W103.07  ; 出料定位下层左右夹紧手动
OUT W143.07  ; 出料定位下层左右夹紧[M]
LD TR0
AND W20.01  ; 2ST-B自动允许输出
OUT TR1
AND D1035.03  ; 2St_出料定位步03 全部松开
OUT W183.06  ; 出料定位下层左右松开[A]
LD TR1
AND D1035.01  ; 2St_出料定位步01前后左右夹紧
AND T0136  ; 出料定位下层前后夹紧位延时
OUT W183.07  ; 出料定位下层左右夹紧[A]
LD TR0
LD W143.06  ; 出料定位下层左右松开[M]
OR W183.06  ; 出料定位下层左右松开[A]
OR 103.06  ; 出料定位下层左右松开输出
ANDLD
ANDNOT W143.07  ; 出料定位下层左右夹紧[M]
ANDNOT W183.07  ; 出料定位下层左右夹紧[A]
LDNOT T0139  ; 出料定位下层左右松开位延时
OR H0.09  ; 气缸保持（1保持）
ANDLD
OUT 103.06  ; 出料定位下层左右松开输出
LD TR0
LD W143.07  ; 出料定位下层左右夹紧[M]
OR W183.07  ; 出料定位下层左右夹紧[A]
OR 103.07  ; 出料定位下层左右夹紧输出
ANDLD
ANDNOT W143.06  ; 出料定位下层左右松开[M]
ANDNOT W183.06  ; 出料定位下层左右松开[A]
LDNOT T0140  ; 出料定位下层左右夹紧位延时
OR H0.09  ; 气缸保持（1保持）
ANDLD
OUT 103.07  ; 出料定位下层左右夹紧输出

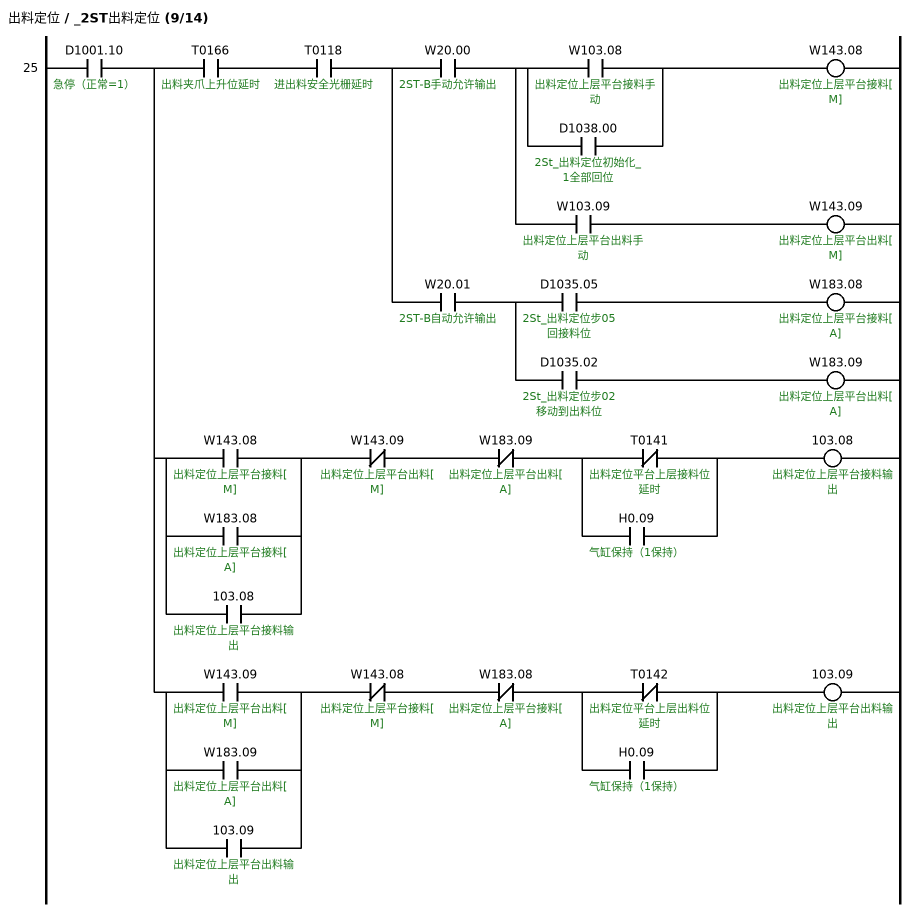
; rung 25
LD D1001.10  ; 急停（正常=1）
OUT TR0
AND T0166  ; 出料夹爪上升位延时
AND T0118  ; 进出料安全光栅延时
OUT TR1
AND W20.00  ; 2ST-B手动允许输出
OUT TR2
LD W103.08  ; 出料定位上层平台接料手动
OR D1038.00  ; 2St_出料定位初始化_1全部回位
ANDLD
OUT W143.08  ; 出料定位上层平台接料[M]
LD TR2
AND W103.09  ; 出料定位上层平台出料手动
OUT W143.09  ; 出料定位上层平台出料[M]
LD TR1
AND W20.01  ; 2ST-B自动允许输出
OUT TR1
AND D1035.05  ; 2St_出料定位步05 回接料位
OUT W183.08  ; 出料定位上层平台接料[A]
LD TR1
AND D1035.02  ; 2St_出料定位步02 移动到出料位
OUT W183.09  ; 出料定位上层平台出料[A]
LD TR0
LD W143.08  ; 出料定位上层平台接料[M]
OR W183.08  ; 出料定位上层平台接料[A]
OR 103.08  ; 出料定位上层平台接料输出
ANDLD
ANDNOT W143.09  ; 出料定位上层平台出料[M]
ANDNOT W183.09  ; 出料定位上层平台出料[A]
LDNOT T0141  ; 出料定位平台上层接料位延时
OR H0.09  ; 气缸保持（1保持）
ANDLD
OUT 103.08  ; 出料定位上层平台接料输出
LD TR0
LD W143.09  ; 出料定位上层平台出料[M]
OR W183.09  ; 出料定位上层平台出料[A]
OR 103.09  ; 出料定位上层平台出料输出
ANDLD
ANDNOT W143.08  ; 出料定位上层平台接料[M]
ANDNOT W183.08  ; 出料定位上层平台接料[A]
LDNOT T0142  ; 出料定位平台上层出料位延时
OR H0.09  ; 气缸保持（1保持）
ANDLD
OUT 103.09  ; 出料定位上层平台出料输出

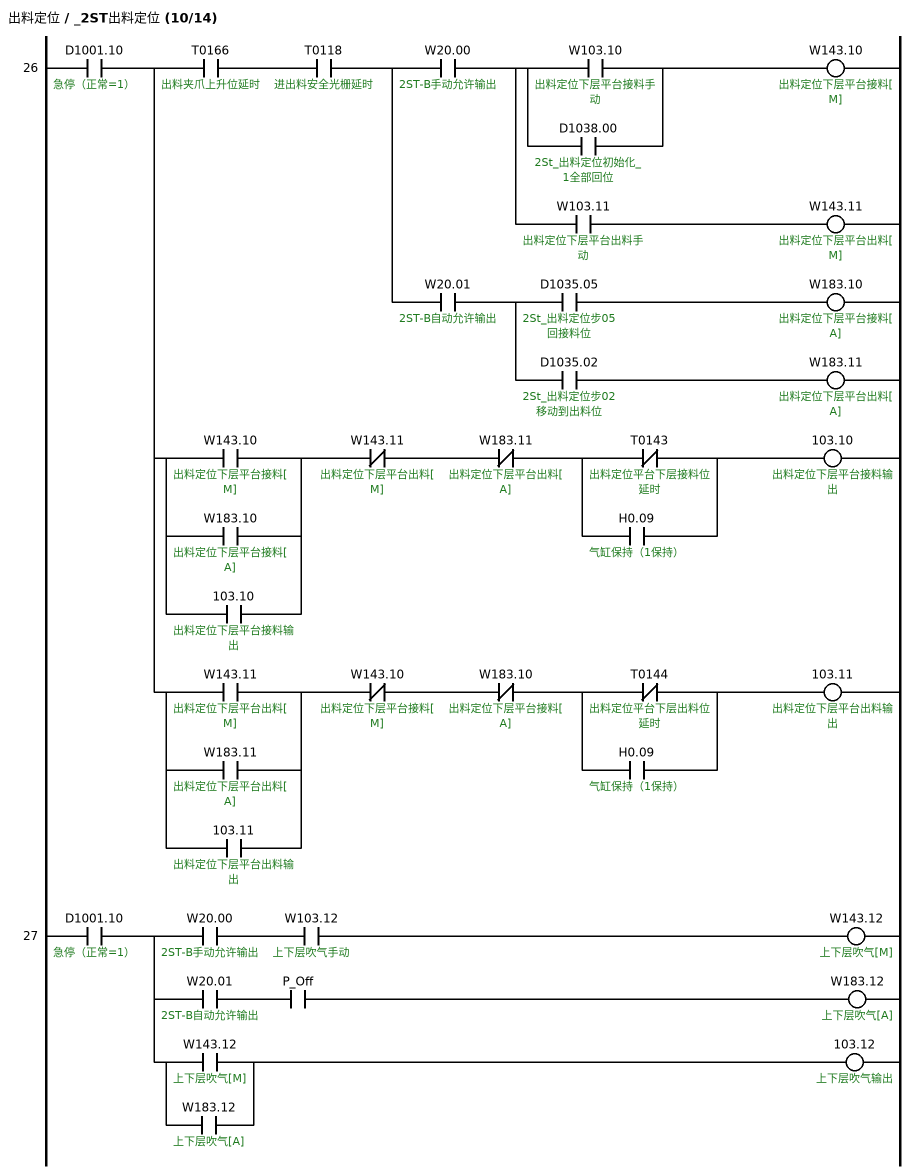
; rung 26
LD D1001.10  ; 急停（正常=1）
OUT TR0
AND T0166  ; 出料夹爪上升位延时
AND T0118  ; 进出料安全光栅延时
OUT TR1
AND W20.00  ; 2ST-B手动允许输出
OUT TR2
LD W103.10  ; 出料定位下层平台接料手动
OR D1038.00  ; 2St_出料定位初始化_1全部回位
ANDLD
OUT W143.10  ; 出料定位下层平台接料[M]
LD TR2
AND W103.11  ; 出料定位下层平台出料手动
OUT W143.11  ; 出料定位下层平台出料[M]
LD TR1
AND W20.01  ; 2ST-B自动允许输出
OUT TR1
AND D1035.05  ; 2St_出料定位步05 回接料位
OUT W183.10  ; 出料定位下层平台接料[A]
LD TR1
AND D1035.02  ; 2St_出料定位步02 移动到出料位
OUT W183.11  ; 出料定位下层平台出料[A]
LD TR0
LD W143.10  ; 出料定位下层平台接料[M]
OR W183.10  ; 出料定位下层平台接料[A]
OR 103.10  ; 出料定位下层平台接料输出
ANDLD
ANDNOT W143.11  ; 出料定位下层平台出料[M]
ANDNOT W183.11  ; 出料定位下层平台出料[A]
LDNOT T0143  ; 出料定位平台下层接料位延时
OR H0.09  ; 气缸保持（1保持）
ANDLD
OUT 103.10  ; 出料定位下层平台接料输出
LD TR0
LD W143.11  ; 出料定位下层平台出料[M]
OR W183.11  ; 出料定位下层平台出料[A]
OR 103.11  ; 出料定位下层平台出料输出
ANDLD
ANDNOT W143.10  ; 出料定位下层平台接料[M]
ANDNOT W183.10  ; 出料定位下层平台接料[A]
LDNOT T0144  ; 出料定位平台下层出料位延时
OR H0.09  ; 气缸保持（1保持）
ANDLD
OUT 103.11  ; 出料定位下层平台出料输出
; rung 27
LD D1001.10  ; 急停（正常=1）
OUT TR0
AND W20.00  ; 2ST-B手动允许输出
AND W103.12  ; 上下层吹气手动
OUT W143.12  ; 上下层吹气[M]
LD TR0
AND W20.01  ; 2ST-B自动允许输出
AND P_Off
OUT W183.12  ; 上下层吹气[A]
LD TR0
LD W143.12  ; 上下层吹气[M]
OR W183.12  ; 上下层吹气[A]
ANDLD
OUT 103.12  ; 上下层吹气输出

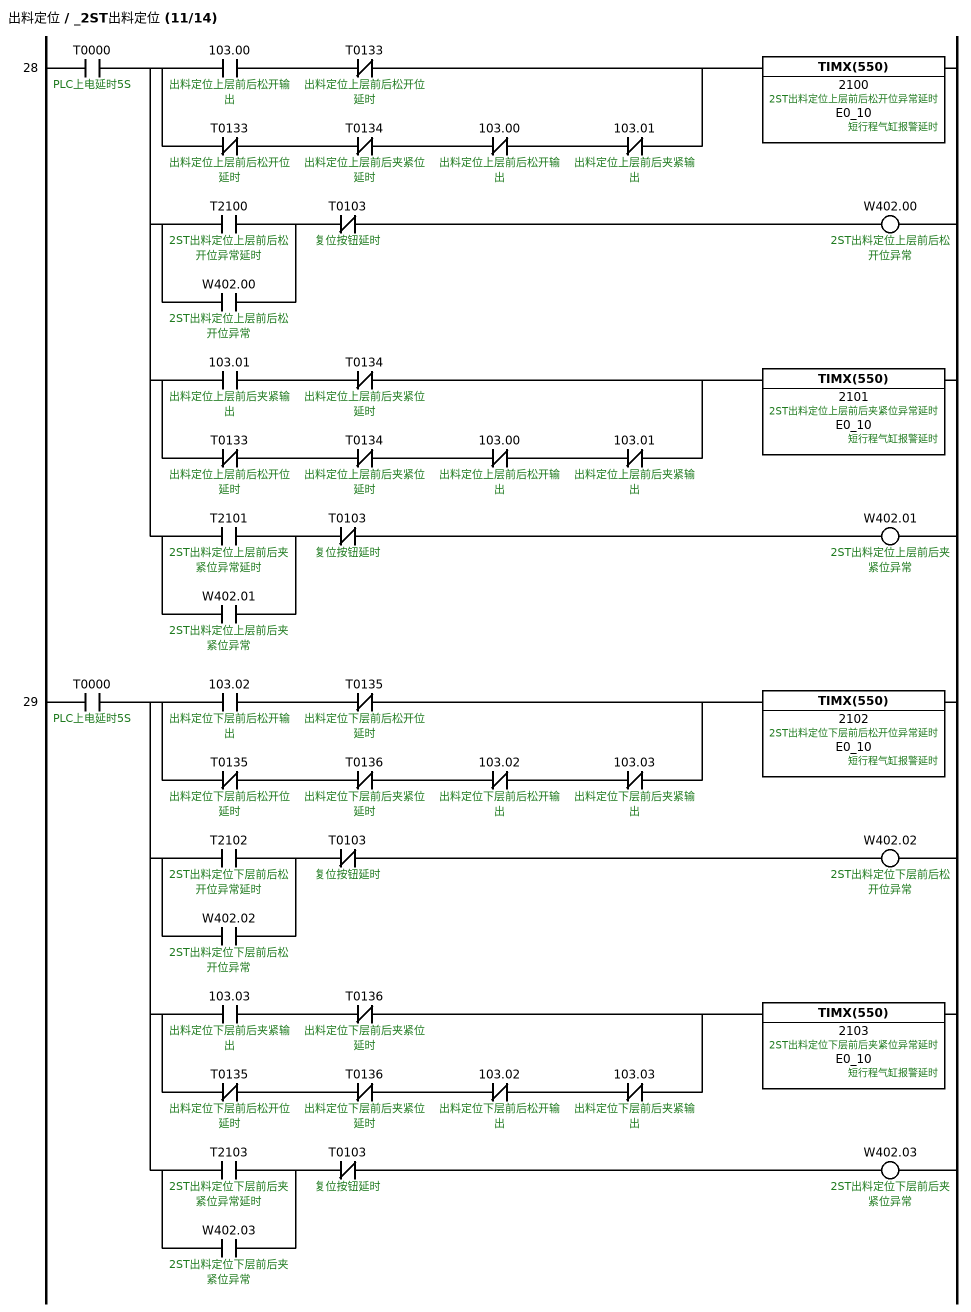
; rung 28
LD T0000  ; PLC上电延时5S
OUT TR0
LD 103.00  ; 出料定位上层前后松开输出
ANDNOT T0133  ; 出料定位上层前后松开位延时
LDNOT T0133  ; 出料定位上层前后松开位延时
ANDNOT T0134  ; 出料定位上层前后夹紧位延时
ANDNOT 103.00  ; 出料定位上层前后松开输出
ANDNOT 103.01  ; 出料定位上层前后夹紧输出
ORLD
ANDLD
TIMX(550) 2100 E0_10  ; 短行程气缸报警延时, 2ST出料定位上层前后松开位异常延时
LD TR0
LD T2100  ; 2ST出料定位上层前后松开位异常延时
OR W402.00  ; 2ST出料定位上层前后松开位异常
ANDLD
ANDNOT T0103  ; 复位按钮延时
OUT W402.00  ; 2ST出料定位上层前后松开位异常
LD TR0
LD 103.01  ; 出料定位上层前后夹紧输出
ANDNOT T0134  ; 出料定位上层前后夹紧位延时
LDNOT T0133  ; 出料定位上层前后松开位延时
ANDNOT T0134  ; 出料定位上层前后夹紧位延时
ANDNOT 103.00  ; 出料定位上层前后松开输出
ANDNOT 103.01  ; 出料定位上层前后夹紧输出
ORLD
ANDLD
TIMX(550) 2101 E0_10  ; 短行程气缸报警延时, 2ST出料定位上层前后夹紧位异常延时
LD TR0
LD T2101  ; 2ST出料定位上层前后夹紧位异常延时
OR W402.01  ; 2ST出料定位上层前后夹紧位异常
ANDLD
ANDNOT T0103  ; 复位按钮延时
OUT W402.01  ; 2ST出料定位上层前后夹紧位异常
; rung 29
LD T0000  ; PLC上电延时5S
OUT TR0
LD 103.02  ; 出料定位下层前后松开输出
ANDNOT T0135  ; 出料定位下层前后松开位延时
LDNOT T0135  ; 出料定位下层前后松开位延时
ANDNOT T0136  ; 出料定位下层前后夹紧位延时
ANDNOT 103.02  ; 出料定位下层前后松开输出
ANDNOT 103.03  ; 出料定位下层前后夹紧输出
ORLD
ANDLD
TIMX(550) 2102 E0_10  ; 短行程气缸报警延时, 2ST出料定位下层前后松开位异常延时
LD TR0
LD T2102  ; 2ST出料定位下层前后松开位异常延时
OR W402.02  ; 2ST出料定位下层前后松开位异常
ANDLD
ANDNOT T0103  ; 复位按钮延时
OUT W402.02  ; 2ST出料定位下层前后松开位异常
LD TR0
LD 103.03  ; 出料定位下层前后夹紧输出
ANDNOT T0136  ; 出料定位下层前后夹紧位延时
LDNOT T0135  ; 出料定位下层前后松开位延时
ANDNOT T0136  ; 出料定位下层前后夹紧位延时
ANDNOT 103.02  ; 出料定位下层前后松开输出
ANDNOT 103.03  ; 出料定位下层前后夹紧输出
ORLD
ANDLD
TIMX(550) 2103 E0_10  ; 短行程气缸报警延时, 2ST出料定位下层前后夹紧位异常延时
LD TR0
LD T2103  ; 2ST出料定位下层前后夹紧位异常延时
OR W402.03  ; 2ST出料定位下层前后夹紧位异常
ANDLD
ANDNOT T0103  ; 复位按钮延时
OUT W402.03  ; 2ST出料定位下层前后夹紧位异常

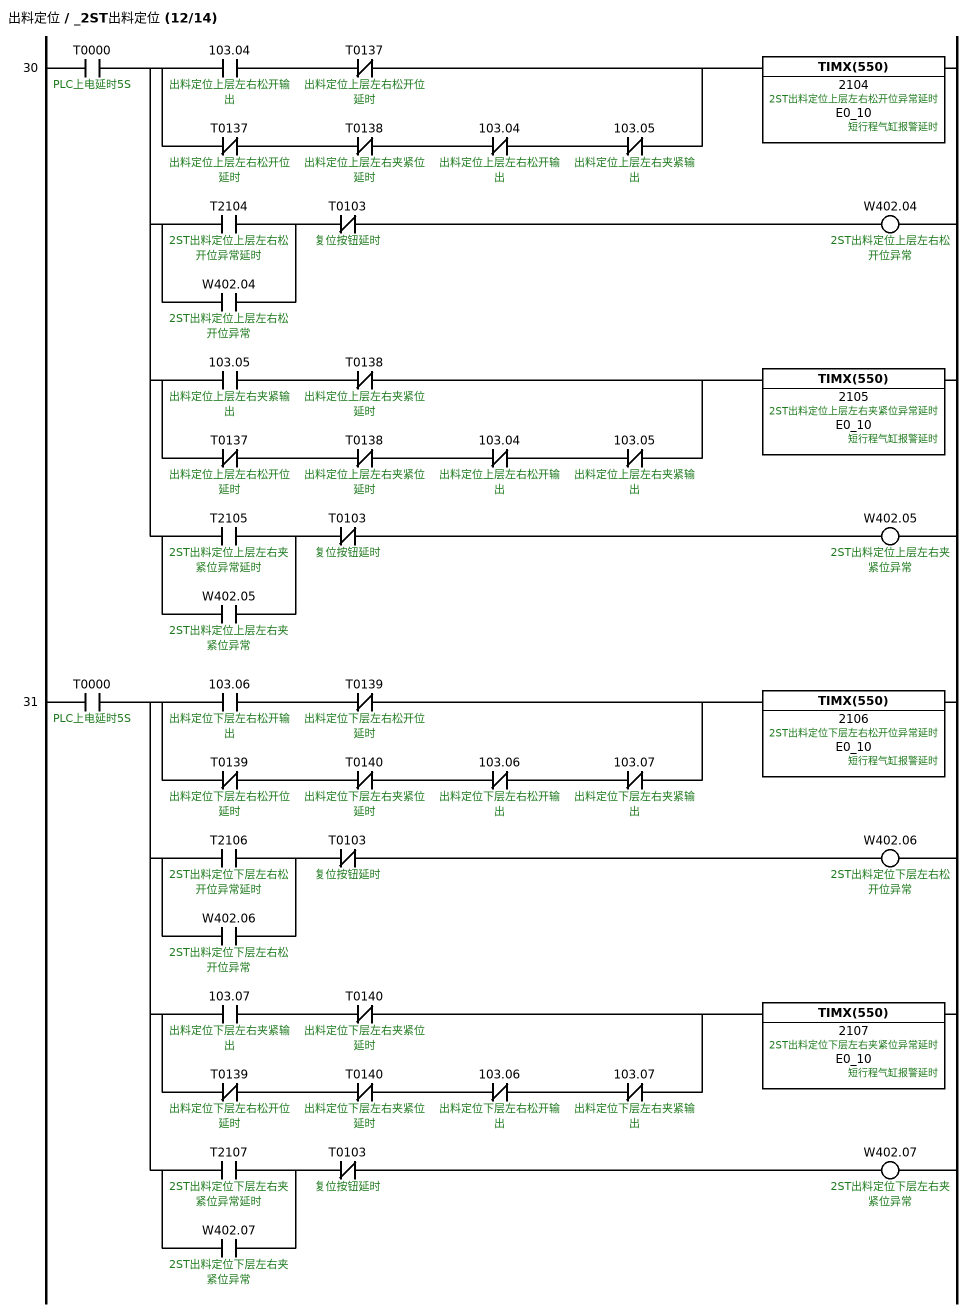
; rung 30
LD T0000  ; PLC上电延时5S
OUT TR0
LD 103.04  ; 出料定位上层左右松开输出
ANDNOT T0137  ; 出料定位上层左右松开位延时
LDNOT T0137  ; 出料定位上层左右松开位延时
ANDNOT T0138  ; 出料定位上层左右夹紧位延时
ANDNOT 103.04  ; 出料定位上层左右松开输出
ANDNOT 103.05  ; 出料定位上层左右夹紧输出
ORLD
ANDLD
TIMX(550) 2104 E0_10  ; 短行程气缸报警延时, 2ST出料定位上层左右松开位异常延时
LD TR0
LD T2104  ; 2ST出料定位上层左右松开位异常延时
OR W402.04  ; 2ST出料定位上层左右松开位异常
ANDLD
ANDNOT T0103  ; 复位按钮延时
OUT W402.04  ; 2ST出料定位上层左右松开位异常
LD TR0
LD 103.05  ; 出料定位上层左右夹紧输出
ANDNOT T0138  ; 出料定位上层左右夹紧位延时
LDNOT T0137  ; 出料定位上层左右松开位延时
ANDNOT T0138  ; 出料定位上层左右夹紧位延时
ANDNOT 103.04  ; 出料定位上层左右松开输出
ANDNOT 103.05  ; 出料定位上层左右夹紧输出
ORLD
ANDLD
TIMX(550) 2105 E0_10  ; 短行程气缸报警延时, 2ST出料定位上层左右夹紧位异常延时
LD TR0
LD T2105  ; 2ST出料定位上层左右夹紧位异常延时
OR W402.05  ; 2ST出料定位上层左右夹紧位异常
ANDLD
ANDNOT T0103  ; 复位按钮延时
OUT W402.05  ; 2ST出料定位上层左右夹紧位异常
; rung 31
LD T0000  ; PLC上电延时5S
OUT TR0
LD 103.06  ; 出料定位下层左右松开输出
ANDNOT T0139  ; 出料定位下层左右松开位延时
LDNOT T0139  ; 出料定位下层左右松开位延时
ANDNOT T0140  ; 出料定位下层左右夹紧位延时
ANDNOT 103.06  ; 出料定位下层左右松开输出
ANDNOT 103.07  ; 出料定位下层左右夹紧输出
ORLD
ANDLD
TIMX(550) 2106 E0_10  ; 短行程气缸报警延时, 2ST出料定位下层左右松开位异常延时
LD TR0
LD T2106  ; 2ST出料定位下层左右松开位异常延时
OR W402.06  ; 2ST出料定位下层左右松开位异常
ANDLD
ANDNOT T0103  ; 复位按钮延时
OUT W402.06  ; 2ST出料定位下层左右松开位异常
LD TR0
LD 103.07  ; 出料定位下层左右夹紧输出
ANDNOT T0140  ; 出料定位下层左右夹紧位延时
LDNOT T0139  ; 出料定位下层左右松开位延时
ANDNOT T0140  ; 出料定位下层左右夹紧位延时
ANDNOT 103.06  ; 出料定位下层左右松开输出
ANDNOT 103.07  ; 出料定位下层左右夹紧输出
ORLD
ANDLD
TIMX(550) 2107 E0_10  ; 短行程气缸报警延时, 2ST出料定位下层左右夹紧位异常延时
LD TR0
LD T2107  ; 2ST出料定位下层左右夹紧位异常延时
OR W402.07  ; 2ST出料定位下层左右夹紧位异常
ANDLD
ANDNOT T0103  ; 复位按钮延时
OUT W402.07  ; 2ST出料定位下层左右夹紧位异常

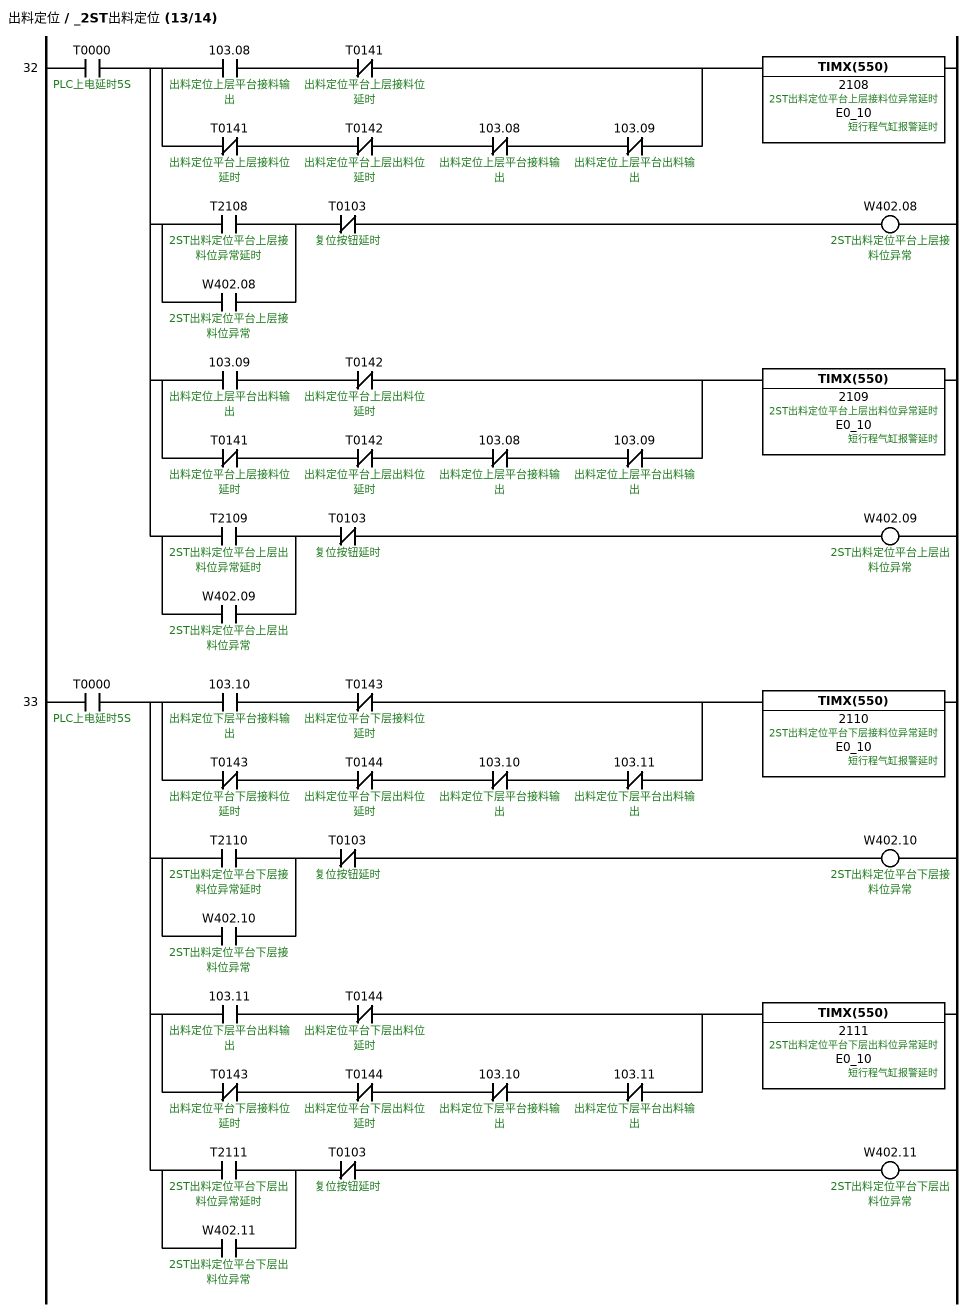
; rung 32
LD T0000  ; PLC上电延时5S
OUT TR0
LD 103.08  ; 出料定位上层平台接料输出
ANDNOT T0141  ; 出料定位平台上层接料位延时
LDNOT T0141  ; 出料定位平台上层接料位延时
ANDNOT T0142  ; 出料定位平台上层出料位延时
ANDNOT 103.08  ; 出料定位上层平台接料输出
ANDNOT 103.09  ; 出料定位上层平台出料输出
ORLD
ANDLD
TIMX(550) 2108 E0_10  ; 短行程气缸报警延时, 2ST出料定位平台上层接料位异常延时
LD TR0
LD T2108  ; 2ST出料定位平台上层接料位异常延时
OR W402.08  ; 2ST出料定位平台上层接料位异常
ANDLD
ANDNOT T0103  ; 复位按钮延时
OUT W402.08  ; 2ST出料定位平台上层接料位异常
LD TR0
LD 103.09  ; 出料定位上层平台出料输出
ANDNOT T0142  ; 出料定位平台上层出料位延时
LDNOT T0141  ; 出料定位平台上层接料位延时
ANDNOT T0142  ; 出料定位平台上层出料位延时
ANDNOT 103.08  ; 出料定位上层平台接料输出
ANDNOT 103.09  ; 出料定位上层平台出料输出
ORLD
ANDLD
TIMX(550) 2109 E0_10  ; 短行程气缸报警延时, 2ST出料定位平台上层出料位异常延时
LD TR0
LD T2109  ; 2ST出料定位平台上层出料位异常延时
OR W402.09  ; 2ST出料定位平台上层出料位异常
ANDLD
ANDNOT T0103  ; 复位按钮延时
OUT W402.09  ; 2ST出料定位平台上层出料位异常
; rung 33
LD T0000  ; PLC上电延时5S
OUT TR0
LD 103.10  ; 出料定位下层平台接料输出
ANDNOT T0143  ; 出料定位平台下层接料位延时
LDNOT T0143  ; 出料定位平台下层接料位延时
ANDNOT T0144  ; 出料定位平台下层出料位延时
ANDNOT 103.10  ; 出料定位下层平台接料输出
ANDNOT 103.11  ; 出料定位下层平台出料输出
ORLD
ANDLD
TIMX(550) 2110 E0_10  ; 短行程气缸报警延时, 2ST出料定位平台下层接料位异常延时
LD TR0
LD T2110  ; 2ST出料定位平台下层接料位异常延时
OR W402.10  ; 2ST出料定位平台下层接料位异常
ANDLD
ANDNOT T0103  ; 复位按钮延时
OUT W402.10  ; 2ST出料定位平台下层接料位异常
LD TR0
LD 103.11  ; 出料定位下层平台出料输出
ANDNOT T0144  ; 出料定位平台下层出料位延时
LDNOT T0143  ; 出料定位平台下层接料位延时
ANDNOT T0144  ; 出料定位平台下层出料位延时
ANDNOT 103.10  ; 出料定位下层平台接料输出
ANDNOT 103.11  ; 出料定位下层平台出料输出
ORLD
ANDLD
TIMX(550) 2111 E0_10  ; 短行程气缸报警延时, 2ST出料定位平台下层出料位异常延时
LD TR0
LD T2111  ; 2ST出料定位平台下层出料位异常延时
OR W402.11  ; 2ST出料定位平台下层出料位异常
ANDLD
ANDNOT T0103  ; 复位按钮延时
OUT W402.11  ; 2ST出料定位平台下层出料位异常

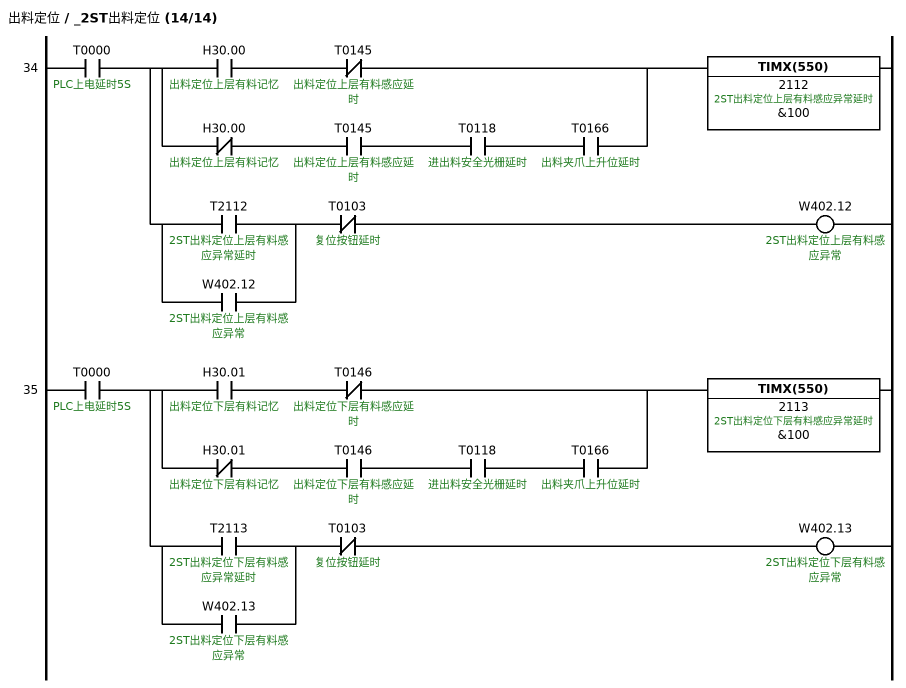
; rung 34
LD T0000  ; PLC上电延时5S
OUT TR0
LD H30.00  ; 出料定位上层有料记忆
ANDNOT T0145  ; 出料定位上层有料感应延时
LDNOT H30.00  ; 出料定位上层有料记忆
AND T0145  ; 出料定位上层有料感应延时
AND T0118  ; 进出料安全光栅延时
AND T0166  ; 出料夹爪上升位延时
ORLD
ANDLD
TIMX(550) 2112 &100  ; 2ST出料定位上层有料感应异常延时
LD TR0
LD T2112  ; 2ST出料定位上层有料感应异常延时
OR W402.12  ; 2ST出料定位上层有料感应异常
ANDLD
ANDNOT T0103  ; 复位按钮延时
OUT W402.12  ; 2ST出料定位上层有料感应异常
; rung 35
LD T0000  ; PLC上电延时5S
OUT TR0
LD H30.01  ; 出料定位下层有料记忆
ANDNOT T0146  ; 出料定位下层有料感应延时
LDNOT H30.01  ; 出料定位下层有料记忆
AND T0146  ; 出料定位下层有料感应延时
AND T0118  ; 进出料安全光栅延时
AND T0166  ; 出料夹爪上升位延时
ORLD
ANDLD
TIMX(550) 2113 &100  ; 2ST出料定位下层有料感应异常延时
LD TR0
LD T2113  ; 2ST出料定位下层有料感应异常延时
OR W402.13  ; 2ST出料定位下层有料感应异常
ANDLD
ANDNOT T0103  ; 复位按钮延时
OUT W402.13  ; 2ST出料定位下层有料感应异常

### Section 复位

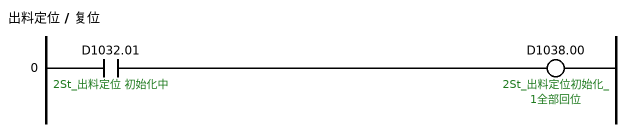
; rung 0
LD D1032.01  ; 2St_出料定位 初始化中
OUT D1038.00  ; 2St_出料定位初始化_1全部回位

### Section 输出

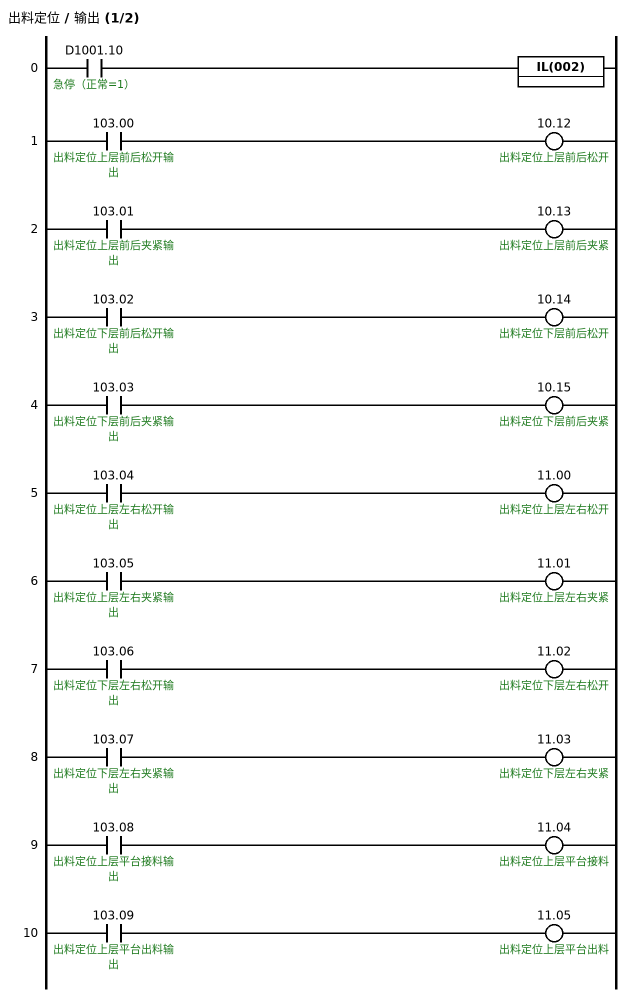
; rung 0
LD D1001.10  ; 急停（正常=1）
IL(002)
; rung 1
LD 103.00  ; 出料定位上层前后松开输出
OUT 10.12  ; 出料定位上层前后松开
; rung 2
LD 103.01  ; 出料定位上层前后夹紧输出
OUT 10.13  ; 出料定位上层前后夹紧
; rung 3
LD 103.02  ; 出料定位下层前后松开输出
OUT 10.14  ; 出料定位下层前后松开
; rung 4
LD 103.03  ; 出料定位下层前后夹紧输出
OUT 10.15  ; 出料定位下层前后夹紧
; rung 5
LD 103.04  ; 出料定位上层左右松开输出
OUT 11.00  ; 出料定位上层左右松开
; rung 6
LD 103.05  ; 出料定位上层左右夹紧输出
OUT 11.01  ; 出料定位上层左右夹紧
; rung 7
LD 103.06  ; 出料定位下层左右松开输出
OUT 11.02  ; 出料定位下层左右松开
; rung 8
LD 103.07  ; 出料定位下层左右夹紧输出
OUT 11.03  ; 出料定位下层左右夹紧
; rung 9
LD 103.08  ; 出料定位上层平台接料输出
OUT 11.04  ; 出料定位上层平台接料
; rung 10
LD 103.09  ; 出料定位上层平台出料输出
OUT 11.05  ; 出料定位上层平台出料

